# B&R Automation Studio project A2019059_Linka_Power_CP (part 47)

#### Main.st - Init, cyclic, exit code
```iecst
PROGRAM _INIT
	(* Insert code here *)
    SKTcpClientTrace_1.Params.IPportClient := 21001;
END_PROGRAM

PROGRAM _CYCLIC

	//Priradenie indexu paletky//
    a:= P3_LeakageTestB.PAR.IndexPaletky;

    //Parametre komunikácie//
    memcpy(ADR(SKTcpClientTrace_1.Params.IPaddrServ),ADR('192.168.122.250'),SIZEOF('192.168.122.250'));

    SKTcpClientTrace_1.Params.IPportServ := 12000;
    SKTcpClientTrace_1.Params.RecvTimeout := 10000;
    SKTcpClientTrace_1();

    //Parametre komunikácie//
    //Vstupy pre server//
    SKTcpClientTrace_1.Params.Packet.type := TRCB_P3_LeakageTestB_ST8B.INPUTS.TYP_Prikazu;
    SKTcpClientTrace_1.Params.Packet.workplace := TRCB_P3_LeakageTestB_ST8B.INPUTS.CisloStanice;
    TRCB_P3_LeakageTestB_ST8B.INPUTS.CisloPaletky:= 'Pal';
    brsstrcat(ADR(TRCB_P3_LeakageTestB_ST8B.INPUTS.CisloPaletky), ADR(P3_LeakageTestB.PAR.IndexPaletky_STRING));
    SKTcpClientTrace_1.Params.Packet.rfid := TRCB_P3_LeakageTestB_ST8B.INPUTS.CisloPaletky;
    SKTcpClientTrace_1.Params.Packet.master := TRCB_P3_LeakageTestB_ST8B.INPUTS.QRkodPowerCP;
    SKTcpClientTrace_1.Params.Packet.dps1:= TRCB_P3_LeakageTestB_ST8B.INPUTS.QRkodFiltra;
    SKTcpClientTrace_1.Params.Packet.dps2:= '';
    SKTcpClientTrace_1.Params.Packet.dps3:= '';
    SKTcpClientTrace_1.Params.Packet.dps4:= '';
    SKTcpClientTrace_1.Params.Packet.dps5:= '';
    SKTcpClientTrace_1.Params.Packet.operator_id := TRCB_P3_LeakageTestB_ST8B.INPUTS.ID_Operatora;
    SKTcpClientTrace_1.Params.Packet.data_report:= TRCB_P3_LeakageTestB_ST8B.INPUTS.Report;
    SKTcpClientTrace_1.Params.Packet.result := TRCB_P3_LeakageTestB_ST8B.INPUTS.StavPaletky;

    //Výstupy zo servera//
    TRCB_P3_LeakageTestB_ST8B.OUTPUTS.TYP_Prikazu:= SKTcpClientTrace_1.Internal.Splitter.out[1];
    TRCB_P3_LeakageTestB_ST8B.OUTPUTS.CisloStanice:= SKTcpClientTrace_1.Internal.Splitter.out[2];
    TRCB_P3_LeakageTestB_ST8B.OUTPUTS.CisloPaletky:= SKTcpClientTrace_1.Internal.Splitter.out[3];
    IF TRCB_P3_LeakageTestB_ST8B.INPUTS.TYP_Prikazu = '0' THEN
        TRCB_P3_LeakageTestB_ST8B.OUTPUTS.CisloEtikety:= SKTcpClientTrace_1.Internal.Splitter.out[4];
    ELSE
        TRCB_P3_LeakageTestB_ST8B.OUTPUTS.QRkodPowerCP:= SKTcpClientTrace_1.Internal.Splitter.out[4];
    END_IF
    TRCB_P3_LeakageTestB_ST8B.OUTPUTS.QRkodFiltra:= SKTcpClientTrace_1.Internal.Splitter.out[5];
    TRCB_P3_LeakageTestB_ST8B.OUTPUTS.ID_Operatora:= SKTcpClientTrace_1.Internal.Splitter.out[10];
    TRCB_P3_LeakageTestB_ST8B.OUTPUTS.DruhCinnostiNaPaletke:= SKTcpClientTrace_1.Internal.Splitter.out[11];
    TRCB_P3_LeakageTestB_ST8B.OUTPUTS.PovolenieCinnostiNaPaletke:= SKTcpClientTrace_1.Internal.Splitter.out[12];

    //Volanie funkcie SequenceControl//
    SequenceControl(SC:= SC_KOM_Server);

    CASE SC_KOM_Server.Step OF

        0:
            SC_KOM_Server.StepName:= '0 - Nulovanie';
            SKTcpClientTrace_1.Cmd.Send:= FALSE;
            SKTcpClientTrace_1.Cmd.Close:= FALSE;
            TRCB_P3_LeakageTestB_ST8B.CMD.VyziadajStavPaletky_TYP1:= FALSE;
            TRCB_P3_LeakageTestB_ST8B.CMD.PriradQRkodFiltra_TYP3:= FALSE;
            TRCB_P3_LeakageTestB_ST8B.CMD.VyziadajCisloEtikety_TYP0:= FALSE;
            TRCB_P3_LeakageTestB_ST8B.CMD.OdosliStavPaletky_TYP2:= FALSE;
            TRCB_P3_LeakageTestB_ST8B.STATUS.KomunikaciaUkoncena:= FALSE;
            TRCB_P3_LeakageTestB_ST8B.STATUS.KomunikaciaError:= FALSE;
            PocetDopytovNaServer:= 0;

            IF SKTcpClientTrace_1.Internal.Step = 0 THEN
                SKTcpClientTrace_1.Enable:= TRUE;
                SC_KOM_Server.ResetStep:= TRUE;
                SC_KOM_Server.Step:= 1;
            ELSIF SKTcpClientTrace_1.Internal.Step = 15 THEN
                SKTcpClientTrace_1.Enable:= TRUE;
                SC_KOM_Server.ResetStep:= TRUE;
                SC_KOM_Server.Step:= 1;
            ELSE
                SKTcpClientTrace_1.Enable:= FALSE;
            END_IF

        1:
            SC_KOM_Server.StepName:= '1 - Rozhodnutie o cinnosti';
            IF TRCB_P3_LeakageTestB_ST8B.CMD.VyziadajStavPaletky_TYP1 THEN
                SC_KOM_Server.Step:= 10;
            ELSIF TRCB_P3_LeakageTestB_ST8B.CMD.PriradQRkodFiltra_TYP3 THEN
                SC_KOM_Server.Step:= 20;
            ELSIF TRCB_P3_LeakageTestB_ST8B.CMD.VyziadajCisloEtikety_TYP0 THEN
                SC_KOM_Server.Step:= 30;
            ELSIF TRCB_P3_LeakageTestB_ST8B.CMD.OdosliStavPaletky_TYP2 THEN
                SC_KOM_Server.Step:= 40;
            END_IF

        10:
            SC_KOM_Server.StepName:= '10 - Vyziadanie stavu paletky - odoslanie dat na server';
            SC_KOM_Server.IdleTime.PT:= T#3s;
            SC_KOM_Server.AlarmTime.PT:= T#10s;
            SC_KOM_Server.AlarmTime.IN:= TRUE;

            TRCB_P3_LeakageTestB_ST8B.INPUTS.TYP_Prikazu:= '1';
            TRCB_P3_LeakageTestB_ST8B.INPUTS.CisloStanice:= 'ST8B';
            TRCB_P3_LeakageTestB_ST8B.INPUTS.CisloPaletky; //Z programu
            TRCB_P3_LeakageTestB_ST8B.INPUTS.QRkodPowerCP:= Paletka[a].PAR.QRkodPowerCP;
            TRCB_P3_LeakageTestB_ST8B.INPUTS.QRkodFiltra:= '';
            TRCB_P3_LeakageTestB_ST8B.INPUTS.ID_Operatora:= Paletka[a].PAR.ID_Operatora;
            TRCB_P3_LeakageTestB_ST8B.INPUTS.Report:= '';
            TRCB_P3_LeakageTestB_ST8B.INPUTS.StavPaletky:= 'OK';
            SKTcpClientTrace_1.Cmd.Send:= TRUE;

            IF SKTcpClientTrace_1.Cmd.Send AND NOT SKTcpClientTrace_1.Status.staReceived AND NOT SKTcpClientTrace_1.Status.staError THEN
                SC_KOM_Server.ResetStep:= TRUE;
                SC_KOM_Server.Step:= 13;
            ELSIF SC_KOM_Server.AlarmTime.Q AND (SKTcpClientTrace_1.Status.staReceived OR SKTcpClientTrace_1.Status.staError) THEN
                PocetDopytovNaServer:= PocetDopytovNaServer + 1;
                SKTcpClientTrace_1.Cmd.Send:= FALSE;
                SC_KOM_Server.ResetStep:= TRUE;
                SC_KOM_Server.Step:= 14;
            END_IF

        13:
            SC_KOM_Server.StepName:= '13 - Vyziadanie stavu paletky - odpoved servera';
            SC_KOM_Server.IdleTime.PT:= T#3s;
            SC_KOM_Server.AlarmTime.PT:= T#20s;
            SC_KOM_Server.AlarmTime.IN:= TRUE;

            IF SKTcpClientTrace_1.Status.staReceived AND
                (TRCB_P3_LeakageTestB_ST8B.OUTPUTS.TYP_Prikazu = TRCB_P3_LeakageTestB_ST8B.INPUTS.TYP_Prikazu) AND
                (TRCB_P3_LeakageTestB_ST8B.OUTPUTS.QRkodPowerCP = TRCB_P3_LeakageTestB_ST8B.INPUTS.QRkodPowerCP) THEN
                TRCB_P3_LeakageTestB_ST8B.STATUS.KomunikaciaUkoncena:= TRUE;
                SC_KOM_Server.ResetStep:= TRUE;
                SC_KOM_Server.Step:= 15;
            ELSIF SC_KOM_Server.AlarmTime.Q THEN
                PocetDopytovNaServer:= PocetDopytovNaServer + 1;
                SC_KOM_Server.ResetStep:= TRUE;
                SC_KOM_Server.Step:= 14;
            END_IF

        14:
            SC_KOM_Server.StepName:= '14 - Vyziadanie stavu paletky - cakam na opatovny dopyt na server';
            SC_KOM_Server.IdleTime.PT:= T#1s;
            SC_KOM_Server.AlarmTime.PT:= T#10s;
            SC_KOM_Server.IdleTime.IN:= TRUE;

            IF PocetDopytovNaServer < 3 THEN
                IF SC_KOM_Server.IdleTime.Q THEN
                    SC_KOM_Server.ResetStep:= TRUE;
                    SC_KOM_Server.Step:= 10;
                END_IF
            ELSE
                TRCB_P3_LeakageTestB_ST8B.STATUS.KomunikaciaError:= TRUE;
                SC_KOM_Server.ResetStep:= TRUE;
                SC_KOM_Server.Step:= 15;
            END_IF

        15:
            SC_KOM_Server.StepName:= '15 - Vyziadanie stavu paletky - cakam na ukoncenie komunikacie';
            SC_KOM_Server.IdleTime.PT:= T#3s;
            SC_KOM_Server.AlarmTime.PT:= T#10s;

            IF NOT TRCB_P3_LeakageTestB_ST8B.CMD.VyziadajStavPaletky_TYP1 THEN
                SC_KOM_Server.ResetStep:= TRUE;
                SC_KOM_Server.Step:= 0;
            END_IF

        20:
            SC_KOM_Server.StepName:= '20 - Priradenie QR kodu - odoslanie dat na server';
            SC_KOM_Server.IdleTime.PT:= T#3s;
            SC_KOM_Server.AlarmTime.PT:= T#10s;

            TRCB_P3_LeakageTestB_ST8B.INPUTS.TYP_Prikazu:= '3';
            TRCB_P3_LeakageTestB_ST8B.INPUTS.CisloStanice:= 'ST8B';
            TRCB_P3_LeakageTestB_ST8B.INPUTS.CisloPaletky;
            TRCB_P3_LeakageTestB_ST8B.INPUTS.QRkodPowerCP:= Paletka[a].PAR.QRkodPowerCP;
            TRCB_P3_LeakageTestB_ST8B.INPUTS.QRkodFiltra:= '';
            TRCB_P3_LeakageTestB_ST8B.INPUTS.ID_Operatora:= Paletka[a].PAR.ID_Operatora;
            TRCB_P3_LeakageTestB_ST8B.INPUTS.Report:= '';
            TRCB_P3_LeakageTestB_ST8B.INPUTS.StavPaletky:= 'OK';
            SKTcpClientTrace_1.Cmd.Send:= TRUE;

            IF SKTcpClientTrace_1.Cmd.Send AND NOT SKTcpClientTrace_1.Status.staReceived AND NOT SKTcpClientTrace_1.Status.staError THEN
                SC_KOM_Server.ResetStep:= TRUE;
                SC_KOM_Server.Step:= 23;
            END_IF

        23:
            SC_KOM_Server.StepName:= '23 - Priradenie QR kodu - odpoved servera';
            SC_KOM_Server.IdleTime.PT:= T#3s;
            SC_KOM_Server.AlarmTime.PT:= T#20s;
            SC_KOM_Server.AlarmTime.IN:= TRUE;

            IF SKTcpClientTrace_1.Status.staReceived AND
                (TRCB_P3_LeakageTestB_ST8B.OUTPUTS.TYP_Prikazu = TRCB_P3_LeakageTestB_ST8B.INPUTS.TYP_Prikazu) AND
                (TRCB_P3_LeakageTestB_ST8B.OUTPUTS.QRkodPowerCP = TRCB_P3_LeakageTestB_ST8B.INPUTS.QRkodPowerCP) THEN
                TRCB_P3_LeakageTestB_ST8B.STATUS.KomunikaciaUkoncena:= TRUE;
                SC_KOM_Server.ResetStep:= TRUE;
                SC_KOM_Server.Step:= 25;
            ELSIF SC_KOM_Server.AlarmTime.Q THEN
                TRCB_P3_LeakageTestB_ST8B.STATUS.KomunikaciaError:= TRUE;
                SC_KOM_Server.ResetStep:= TRUE;
                SC_KOM_Server.Step:= 25;
            END_IF

        25:
            SC_KOM_Server.StepName:= '25 - Vyziadanie stavu paletky - cakam na ukoncenie komunikacie';
            SC_KOM_Server.IdleTime.PT:= T#3s;
            SC_KOM_Server.AlarmTime.PT:= T#10s;

            IF NOT TRCB_P3_LeakageTestB_ST8B.CMD.PriradQRkodFiltra_TYP3 THEN
                SC_KOM_Server.ResetStep:= TRUE;
                SC_KOM_Server.Step:= 0;
            END_IF

        30:
            SC_KOM_Server.StepName:= '30 - Vyziadanie serioveho cisla - odoslanie dat na server';
            SC_KOM_Server.IdleTime.PT:= T#3s;
            SC_KOM_Server.AlarmTime.PT:= T#10s;

            TRCB_P3_LeakageTestB_ST8B.INPUTS.TYP_Prikazu:= '0';
            TRCB_P3_LeakageTestB_ST8B.INPUTS.CisloStanice:= 'ST8B';
            TRCB_P3_LeakageTestB_ST8B.INPUTS.CisloPaletky;
            TRCB_P3_LeakageTestB_ST8B.INPUTS.QRkodPowerCP:= '';
            TRCB_P3_LeakageTestB_ST8B.INPUTS.QRkodFiltra:= '';
            TRCB_P3_LeakageTestB_ST8B.INPUTS.ID_Operatora:= 'E2';
            TRCB_P3_LeakageTestB_ST8B.INPUTS.Report:= '';
            TRCB_P3_LeakageTestB_ST8B.INPUTS.StavPaletky:= 'OK';
            SKTcpClientTrace_1.Cmd.Send:= TRUE;

            IF SKTcpClientTrace_1.Cmd.Send AND NOT SKTcpClientTrace_1.Status.staReceived AND NOT SKTcpClientTrace_1.Status.staError THEN
                SC_KOM_Server.ResetStep:= TRUE;
                SC_KOM_Server.Step:= 33;
            END_IF

        33:
            SC_KOM_Server.StepName:= '33 - Vyziadanie serioveho cisla - odpoved servera';
            SC_KOM_Server.IdleTime.PT:= T#3s;
            SC_KOM_Server.AlarmTime.PT:= T#20s;
            SC_KOM_Server.AlarmTime.IN:= TRUE;

            IF SKTcpClientTrace_1.Status.staReceived AND
                (TRCB_P3_LeakageTestB_ST8B.OUTPUTS.TYP_Prikazu = TRCB_P3_LeakageTestB_ST8B.INPUTS.TYP_Prikazu) THEN
                TRCB_P3_LeakageTestB_ST8B.STATUS.KomunikaciaUkoncena:= TRUE;
                SC_KOM_Server.ResetStep:= TRUE;
                SC_KOM_Server.Step:= 35;
            ELSIF SC_KOM_Server.AlarmTime.Q THEN
                TRCB_P3_LeakageTestB_ST8B.STATUS.KomunikaciaError:= TRUE;
                SC_KOM_Server.ResetStep:= TRUE;
                SC_KOM_Server.Step:= 35;
            END_IF

        35:
            SC_KOM_Server.StepName:= '35 - Vyziadanie serioveho cisla - cakam na ukoncenie komunikacie';
            SC_KOM_Server.IdleTime.PT:= T#3s;
            SC_KOM_Server.AlarmTime.PT:= T#10s;

            IF NOT TRCB_P3_LeakageTestB_ST8B.CMD.VyziadajCisloEtikety_TYP0 THEN
                SC_KOM_Server.ResetStep:= TRUE;
                SC_KOM_Server.Step:= 0;
            END_IF

        40:
            SC_KOM_Server.StepName:= '40 - Odoslanie stavu paletky - odoslanie dat na server';
            SC_KOM_Server.IdleTime.PT:= T#3s;
            SC_KOM_Server.AlarmTime.PT:= T#20s;
            SC_KOM_Server.AlarmTime.IN:= TRUE;

            //Vytvorenie spravy pre report//
            IF NOT SC_KOM_Server.Switch1 THEN
                brsmemset(ADR(Report),0,SIZEOF(Report));
                brsmemset(ADR(TRCB_P3_LeakageTestB_ST8B.INPUTS.Report), 0, SIZEOF(TRCB_P3_LeakageTestB_ST8B.INPUTS.Report));

				//Čas plnenia//
                Report[0].PoradoveCislo:= '1';
                Report[0].Popis:= 'StanicaB_CasPlnenia';
                Report[0].FormatHodnoty:= '1';
                Report[0].Tolerancia_MIN_Hodnota:= '';
                Report[0].Tolerancia_MAX_Hodnota:= '';
                Report[0].Nominal:= '';
                Report[0].Tolerancia_MIN_Jednotky:= '';
                Report[0].Tolerancia_MAX_Jednotky:= '';
                Report[0].NameranaHodnota:= Reports.LeakageTest.CasPlnenia.StanicaB;
                Report[0].NameranaHodnota_Jednotky:= 's';
                Report[0].VyslednyResult:= Reports.LeakageTest.VyslednyReport.StanicaB;
                SKTcpClientNewCsvEntry(Report[0].PoradoveCislo,Report[0].Popis,Report[0].FormatHodnoty,Report[0].Tolerancia_MIN_Hodnota,Report[0].Tolerancia_MAX_Hodnota,Report[0].Nominal,Report[0].Tolerancia_MIN_Jednotky,Report[0].Tolerancia_MAX_Jednotky,Report[0].NameranaHodnota,Report[0].NameranaHodnota_Jednotky,Report[0].VyslednyResult, ADR(TRCB_P3_LeakageTestB_ST8B.INPUTS.Report));

                //Čas stabilizacie//
                Report[1].PoradoveCislo:= '2';
                Report[1].Popis:= 'StanicaB_CasStabilizacie';
                Report[1].FormatHodnoty:= '1';
                Report[1].Tolerancia_MIN_Hodnota:= '';
                Report[1].Tolerancia_MAX_Hodnota:= '';
                Report[1].Nominal:= '';
                Report[1].Tolerancia_MIN_Jednotky:= '';
                Report[1].Tolerancia_MAX_Jednotky:= '';
                Report[1].NameranaHodnota:= Reports.LeakageTest.CasStabilizacie.StanicaB;
                Report[1].NameranaHodnota_Jednotky:= 's';
                Report[1].VyslednyResult:= Reports.LeakageTest.VyslednyReport.StanicaB;
                SKTcpClientNewCsvEntry(Report[1].PoradoveCislo,Report[1].Popis,Report[1].FormatHodnoty,Report[1].Tolerancia_MIN_Hodnota,Report[1].Tolerancia_MAX_Hodnota,Report[1].Nominal,Report[1].Tolerancia_MIN_Jednotky,Report[1].Tolerancia_MAX_Jednotky,Report[1].NameranaHodnota,Report[1].NameranaHodnota_Jednotky,Report[1].VyslednyResult, ADR(TRCB_P3_LeakageTestB_ST8B.INPUTS.Report));

                //Tlak plnenia//
                Report[2].PoradoveCislo:= '3';
                Report[2].Popis:= 'StanicaB_TlakPlnenia';
                Report[2].FormatHodnoty:= '1';
                Report[2].Tolerancia_MIN_Hodnota:= '';
                Report[2].Tolerancia_MAX_Hodnota:= '';
                Report[2].Nominal:= '';
                Report[2].Tolerancia_MIN_Jednotky:= '';
                Report[2].Tolerancia_MAX_Jednotky:= '';
                Report[2].NameranaHodnota:= Reports.LeakageTest.TlakPlnenia.StanicaB;
                Report[2].NameranaHodnota_Jednotky:= 'mBar';
                Report[2].VyslednyResult:= Reports.LeakageTest.VyslednyReport.StanicaB;
                SKTcpClientNewCsvEntry(Report[2].PoradoveCislo,Report[2].Popis,Report[2].FormatHodnoty,Report[2].Tolerancia_MIN_Hodnota,Report[2].Tolerancia_MAX_Hodnota,Report[2].Nominal,Report[2].Tolerancia_MIN_Jednotky,Report[2].Tolerancia_MAX_Jednotky,Report[2].NameranaHodnota,Report[2].NameranaHodnota_Jednotky,Report[2].VyslednyResult, ADR(TRCB_P3_LeakageTestB_ST8B.INPUTS.Report));

                //Tlak prítlaku//
                Report[3].PoradoveCislo:= '4';
                Report[3].Popis:= 'StanicaB_TlakPritlaku';
                Report[3].FormatHodnoty:= '1';
                Report[3].Tolerancia_MIN_Hodnota:= Reports.LeakageTest.ToleranciaPritlaku_MIN.StanicaB;
                Report[3].Tolerancia_MAX_Hodnota:= Reports.LeakageTest.ToleranciaPritlaku_MAX.StanicaB;
                Report[3].Nominal:= '';
                Report[3].Tolerancia_MIN_Jednotky:= 'Bar';
                Report[3].Tolerancia_MAX_Jednotky:= 'Bar';
                Report[3].NameranaHodnota:= Reports.LeakageTest.TlakPritlaku.StanicaB;
                Report[3].NameranaHodnota_Jednotky:= 'Bar';
                Report[3].VyslednyResult:= Reports.LeakageTest.VyslednyReport.StanicaB;
                SKTcpClientNewCsvEntry(Report[3].PoradoveCislo,Report[3].Popis,Report[3].FormatHodnoty,Report[3].Tolerancia_MIN_Hodnota,Report[3].Tolerancia_MAX_Hodnota,Report[3].Nominal,Report[3].Tolerancia_MIN_Jednotky,Report[3].Tolerancia_MAX_Jednotky,Report[3].NameranaHodnota,Report[3].NameranaHodnota_Jednotky,Report[3].VyslednyResult, ADR(TRCB_P3_LeakageTestB_ST8B.INPUTS.Report));

                //Tlak úniku//
                Report[4].PoradoveCislo:= '5';
                Report[4].Popis:= 'StanicaB_TlakUniku';
                Report[4].FormatHodnoty:= '1';
                Report[4].Tolerancia_MIN_Hodnota:= Reports.LeakageTest.ToleranciaTlakUniku_MIN.StanicaB;
                Report[4].Tolerancia_MAX_Hodnota:= Reports.LeakageTest.ToleranciaTlakUniku_MAX.StanicaB;
                Report[4].Nominal:= '';
                Report[4].Tolerancia_MIN_Jednotky:= 'Pa';
                Report[4].Tolerancia_MAX_Jednotky:= 'Pa';
                Report[4].NameranaHodnota:= Reports.LeakageTest.TlakUniku.StanicaB;
                Report[4].NameranaHodnota_Jednotky:= 'Pa';
                Report[4].VyslednyResult:= Reports.LeakageTest.VyslednyReport.StanicaB;
                SKTcpClientNewCsvEntry(Report[4].PoradoveCislo,Report[4].Popis,Report[4].FormatHodnoty,Report[4].Tolerancia_MIN_Hodnota,Report[4].Tolerancia_MAX_Hodnota,Report[4].Nominal,Report[4].Tolerancia_MIN_Jednotky,Report[4].Tolerancia_MAX_Jednotky,Report[4].NameranaHodnota,Report[4].NameranaHodnota_Jednotky,Report[4].VyslednyResult, ADR(TRCB_P3_LeakageTestB_ST8B.INPUTS.Report));

                //Tolerancia//
                Report[5].PoradoveCislo:= '6';
                Report[5].Popis:= 'StanicaB_Tolerancia';
                Report[5].FormatHodnoty:= '1';
                Report[5].Tolerancia_MIN_Hodnota:= '';
                Report[5].Tolerancia_MAX_Hodnota:= '';
                Report[5].Nominal:= '';
                Report[5].Tolerancia_MIN_Jednotky:= '';
                Report[5].Tolerancia_MAX_Jednotky:= '';
                Report[5].NameranaHodnota:= Reports.LeakageTest.Tolerancia.StanicaB;
                Report[5].NameranaHodnota_Jednotky:= 'Pa';
                Report[5].VyslednyResult:= Reports.LeakageTest.VyslednyReport.StanicaB;
                SKTcpClientNewCsvEntry(Report[5].PoradoveCislo,Report[5].Popis,Report[5].FormatHodnoty,Report[5].Tolerancia_MIN_Hodnota,Report[5].Tolerancia_MAX_Hodnota,Report[5].Nominal,Report[5].Tolerancia_MIN_Jednotky,Report[5].Tolerancia_MAX_Jednotky,Report[5].NameranaHodnota,Report[5].NameranaHodnota_Jednotky,Report[5].VyslednyResult, ADR(TRCB_P3_LeakageTestB_ST8B.INPUTS.Report));

                SC_KOM_Server.Switch1:= TRUE;
            END_IF

            TRCB_P3_LeakageTestB_ST8B.INPUTS.TYP_Prikazu:= '2';
            TRCB_P3_LeakageTestB_ST8B.INPUTS.CisloStanice:= 'ST8B';
            TRCB_P3_LeakageTestB_ST8B.INPUTS.CisloPaletky;
            TRCB_P3_LeakageTestB_ST8B.INPUTS.QRkodPowerCP:= Paletka[a].PAR.QRkodPowerCP;
            TRCB_P3_LeakageTestB_ST8B.INPUTS.QRkodFiltra:= '';
            TRCB_P3_LeakageTestB_ST8B.INPUTS.ID_Operatora:= Paletka[a].PAR.ID_Operatora;
            TRCB_P3_LeakageTestB_ST8B.INPUTS.StavPaletky:= Paletka[a].PAR.StavPowerCP;
            SKTcpClientTrace_1.Cmd.Send:= TRUE;

            IF SKTcpClientTrace_1.Cmd.Send AND NOT SKTcpClientTrace_1.Status.staReceived AND NOT SKTcpClientTrace_1.Status.staError THEN
                SC_KOM_Server.ResetStep:= TRUE;
                SC_KOM_Server.Step:= 43;
            ELSIF SC_KOM_Server.AlarmTime.Q AND (SKTcpClientTrace_1.Status.staReceived OR SKTcpClientTrace_1.Status.staError) THEN
                PocetDopytovNaServer:= PocetDopytovNaServer + 1;
                SC_KOM_Server.ResetStep:= TRUE;
                SC_KOM_Server.Step:= 44;
            END_IF

        43:
            SC_KOM_Server.StepName:= '43 - Odoslanie stavu paletky - odpoved servera';
            SC_KOM_Server.IdleTime.PT:= T#3s;
            SC_KOM_Server.AlarmTime.PT:= T#20s;
            SC_KOM_Server.AlarmTime.IN:= TRUE;

            IF SKTcpClientTrace_1.Status.staReceived AND
                (TRCB_P3_LeakageTestB_ST8B.OUTPUTS.TYP_Prikazu = TRCB_P3_LeakageTestB_ST8B.INPUTS.TYP_Prikazu) AND
                (TRCB_P3_LeakageTestB_ST8B.OUTPUTS.QRkodPowerCP = TRCB_P3_LeakageTestB_ST8B.INPUTS.QRkodPowerCP) THEN
                TRCB_P3_LeakageTestB_ST8B.STATUS.KomunikaciaUkoncena:= TRUE;
                SC_KOM_Server.ResetStep:= TRUE;
                SC_KOM_Server.Step:= 45;
            ELSIF SC_KOM_Server.AlarmTime.Q THEN
                PocetDopytovNaServer:= PocetDopytovNaServer + 1;
                SC_KOM_Server.ResetStep:= TRUE;
                SC_KOM_Server.Step:= 44;
            END_IF

        44:
            SC_KOM_Server.StepName:= '44 - Odoslanie stavu paletky - cakam na opatovny dopyt na server';
            SC_KOM_Server.IdleTime.PT:= T#1s;
            SC_KOM_Server.AlarmTime.PT:= T#10s;
            SC_KOM_Server.IdleTime.IN:= TRUE;
            SKTcpClientTrace_1.Cmd.Send:= FALSE;

            IF PocetDopytovNaServer < 3 THEN
                IF SC_KOM_Server.IdleTime.Q THEN
                    SC_KOM_Server.ResetStep:= TRUE;
                    SC_KOM_Server.Step:= 40;
                END_IF
            ELSE
                TRCB_P3_LeakageTestB_ST8B.STATUS.KomunikaciaError:= TRUE;
                SC_KOM_Server.ResetStep:= TRUE;
                SC_KOM_Server.Step:= 45;
            END_IF

        45:
            SC_KOM_Server.StepName:= '45 - Odoslanie stavu paletky - cakam na ukoncenie komunikacie';
            SC_KOM_Server.IdleTime.PT:= T#3s;
            SC_KOM_Server.AlarmTime.PT:= T#10s;

            IF NOT TRCB_P3_LeakageTestB_ST8B.CMD.OdosliStavPaletky_TYP2 THEN
                SC_KOM_Server.ResetStep:= TRUE;
                SC_KOM_Server.Step:= 0;
            END_IF

    END_CASE

END_PROGRAM

PROGRAM _EXIT
	(* Insert code here *)

END_PROGRAM
```

#### Types.typ - Local data types
```iecst
TYPE
	Report_typ : 	STRUCT
		PoradoveCislo : STRING[2]; (*IDstep - Poradové čislo reportu*)
		Popis : STRING[100]; (*Description - Popis*)
		FormatHodnoty : STRING[2]; (*TypValue - Format zaslané hodnoty  1- Číslo, 2 - Znak*)
		Tolerancia_MIN_Hodnota : STRING[10]; (*MinTol - Minimálna tolerancia meranej veličiny*)
		Tolerancia_MAX_Hodnota : STRING[10]; (*MaxTol - Maximálna tolerancia meranej veličiny*)
		Nominal : STRING[10]; (*Nom - Ak jezvolený formát string tak tu zadáme OK inak je prazdna*)
		Tolerancia_MIN_Jednotky : STRING[10]; (*MinEle - Jednotky minimálnej tolerancie veličiny*)
		Tolerancia_MAX_Jednotky : STRING[10]; (*MaxEle - Jednotky maximálnej tolerancie veličiny*)
		NameranaHodnota : STRING[10]; (*Value - Namerana hodnota veličiny, ak su kamery tak bude hodnota OK alebo NG*)
		NameranaHodnota_Jednotky : STRING[10]; (*ValEle - Jednotky nameranej veličiny*)
		VyslednyResult : STRING[5]; (*Result - Výsledný result  PASS, FAIL, SKIP*)
	END_STRUCT;
END_TYPE
```

#### Variables.var - Local variables
```iecst
VAR
	SC_KOM_Server : SequenceControlTyp;
	SKTcpClientTrace_1 : SKTcpClientTrace;
	a : USINT;
	Report : ARRAY[0..50] OF Report_typ;
	PocetDopytovNaServer : USINT;
END_VAR
```

### Program Logical/TracebilitySystem/P4_Etiketovacka_ST9 (IEC)

#### Main.st - Init, cyclic, exit code
```iecst
PROGRAM _INIT
	(* Insert code here *)
    SKTcpClientTrace_1.Params.IPportClient := 22000;
END_PROGRAM

PROGRAM _CYCLIC

	//Priradenie indexu paletky//
    a:= P4_Etiketovacka.PAR.IndexPaletky;

    //Parametre komunikácie//
    memcpy(ADR(SKTcpClientTrace_1.Params.IPaddrServ),ADR('192.168.122.250'),SIZEOF('192.168.122.250'));

    SKTcpClientTrace_1.Params.IPportServ := 12000;
    SKTcpClientTrace_1.Params.RecvTimeout := 10000;
    SKTcpClientTrace_1();

    //Parametre komunikácie//
    //Vstupy pre server//
    SKTcpClientTrace_1.Params.Packet.type := TRCB_P4_Etiketovacka_ST9.INPUTS.TYP_Prikazu;
    SKTcpClientTrace_1.Params.Packet.workplace := TRCB_P4_Etiketovacka_ST9.INPUTS.CisloStanice;
    TRCB_P4_Etiketovacka_ST9.INPUTS.CisloPaletky:= 'Pal';
    brsstrcat(ADR(TRCB_P4_Etiketovacka_ST9.INPUTS.CisloPaletky), ADR(P4_Etiketovacka.PAR.IndexPaletky_STRING));
    SKTcpClientTrace_1.Params.Packet.rfid := TRCB_P4_Etiketovacka_ST9.INPUTS.CisloPaletky;
    SKTcpClientTrace_1.Params.Packet.master := TRCB_P4_Etiketovacka_ST9.INPUTS.QRkodPowerCP;
    SKTcpClientTrace_1.Params.Packet.dps1:= TRCB_P4_Etiketovacka_ST9.INPUTS.QRkodFiltra;
    SKTcpClientTrace_1.Params.Packet.dps2:= '';
    SKTcpClientTrace_1.Params.Packet.dps3:= '';
    SKTcpClientTrace_1.Params.Packet.dps4:= '';
    SKTcpClientTrace_1.Params.Packet.dps5:= '';
    SKTcpClientTrace_1.Params.Packet.operator_id := TRCB_P4_Etiketovacka_ST9.INPUTS.ID_Operatora;
    SKTcpClientTrace_1.Params.Packet.data_report:= TRCB_P4_Etiketovacka_ST9.INPUTS.Report;
    SKTcpClientTrace_1.Params.Packet.result := TRCB_P4_Etiketovacka_ST9.INPUTS.StavPaletky;

    //Výstupy zo servera//
    TRCB_P4_Etiketovacka_ST9.OUTPUTS.TYP_Prikazu:= SKTcpClientTrace_1.Internal.Splitter.out[1];
    TRCB_P4_Etiketovacka_ST9.OUTPUTS.CisloStanice:= SKTcpClientTrace_1.Internal.Splitter.out[2];
    TRCB_P4_Etiketovacka_ST9.OUTPUTS.CisloPaletky:= SKTcpClientTrace_1.Internal.Splitter.out[3];
    IF TRCB_P4_Etiketovacka_ST9.INPUTS.TYP_Prikazu = '0' THEN
        TRCB_P4_Etiketovacka_ST9.OUTPUTS.CisloEtikety:= SKTcpClientTrace_1.Internal.Splitter.out[4];
    ELSE
        TRCB_P4_Etiketovacka_ST9.OUTPUTS.QRkodPowerCP:= SKTcpClientTrace_1.Internal.Splitter.out[4];
    END_IF
    TRCB_P4_Etiketovacka_ST9.OUTPUTS.QRkodFiltra:= SKTcpClientTrace_1.Internal.Splitter.out[5];
    TRCB_P4_Etiketovacka_ST9.OUTPUTS.ID_Operatora:= SKTcpClientTrace_1.Internal.Splitter.out[10];
    TRCB_P4_Etiketovacka_ST9.OUTPUTS.DruhCinnostiNaPaletke:= SKTcpClientTrace_1.Internal.Splitter.out[11];
    TRCB_P4_Etiketovacka_ST9.OUTPUTS.PovolenieCinnostiNaPaletke:= SKTcpClientTrace_1.Internal.Splitter.out[12];

    //Volanie funkcie SequenceControl//
    SequenceControl(SC:= SC_KOM_Server);

    CASE SC_KOM_Server.Step OF

        0:
            SC_KOM_Server.StepName:= '0 - Nulovanie';
            SKTcpClientTrace_1.Cmd.Send:= FALSE;
            SKTcpClientTrace_1.Cmd.Close:= FALSE;
            TRCB_P4_Etiketovacka_ST9.CMD.VyziadajStavPaletky_TYP1:= FALSE;
            TRCB_P4_Etiketovacka_ST9.CMD.PriradQRkodFiltra_TYP3:= FALSE;
            TRCB_P4_Etiketovacka_ST9.CMD.VyziadajCisloEtikety_TYP0:= FALSE;
            TRCB_P4_Etiketovacka_ST9.CMD.OdosliStavPaletky_TYP2:= FALSE;
            TRCB_P4_Etiketovacka_ST9.STATUS.KomunikaciaUkoncena:= FALSE;
            TRCB_P4_Etiketovacka_ST9.STATUS.KomunikaciaError:= FALSE;
            PocetDopytovNaServer:= 0;

            IF SKTcpClientTrace_1.Internal.Step = 0 THEN
                SKTcpClientTrace_1.Enable:= TRUE;
                SC_KOM_Server.ResetStep:= TRUE;
                SC_KOM_Server.Step:= 1;
            ELSIF SKTcpClientTrace_1.Internal.Step = 15 THEN
                SKTcpClientTrace_1.Enable:= TRUE;
                SC_KOM_Server.ResetStep:= TRUE;
                SC_KOM_Server.Step:= 1;
            ELSE
                SKTcpClientTrace_1.Enable:= FALSE;
            END_IF

        1:
            SC_KOM_Server.StepName:= '1 - Rozhodnutie o cinnosti';
            IF TRCB_P4_Etiketovacka_ST9.CMD.VyziadajStavPaletky_TYP1 THEN
                SC_KOM_Server.Step:= 10;
            ELSIF TRCB_P4_Etiketovacka_ST9.CMD.PriradQRkodFiltra_TYP3 THEN
                SC_KOM_Server.Step:= 20;
            ELSIF TRCB_P4_Etiketovacka_ST9.CMD.VyziadajCisloEtikety_TYP0 THEN
                SC_KOM_Server.Step:= 30;
            ELSIF TRCB_P4_Etiketovacka_ST9.CMD.OdosliStavPaletky_TYP2 THEN
                SC_KOM_Server.Step:= 40;
            END_IF

        10:
            SC_KOM_Server.StepName:= '10 - Vyziadanie stavu paletky - odoslanie dat na server';
            SC_KOM_Server.IdleTime.PT:= T#3s;
            SC_KOM_Server.AlarmTime.PT:= T#10s;
            SC_KOM_Server.AlarmTime.IN:= TRUE;

            TRCB_P4_Etiketovacka_ST9.INPUTS.TYP_Prikazu:= '1';
            TRCB_P4_Etiketovacka_ST9.INPUTS.CisloStanice:= 'ST9';
            TRCB_P4_Etiketovacka_ST9.INPUTS.CisloPaletky; //Z programu
            TRCB_P4_Etiketovacka_ST9.INPUTS.QRkodPowerCP:= Paletka[a].PAR.QRkodPowerCP;
            TRCB_P4_Etiketovacka_ST9.INPUTS.QRkodFiltra:= '';
            TRCB_P4_Etiketovacka_ST9.INPUTS.ID_Operatora:= Paletka[a].PAR.ID_Operatora;
            TRCB_P4_Etiketovacka_ST9.INPUTS.Report:= '';
            TRCB_P4_Etiketovacka_ST9.INPUTS.StavPaletky:= 'OK';
            SKTcpClientTrace_1.Cmd.Send:= TRUE;

            IF SKTcpClientTrace_1.Cmd.Send AND NOT SKTcpClientTrace_1.Status.staReceived AND NOT SKTcpClientTrace_1.Status.staError THEN
                SC_KOM_Server.ResetStep:= TRUE;
                SC_KOM_Server.Step:= 13;
            ELSIF SC_KOM_Server.AlarmTime.Q AND (SKTcpClientTrace_1.Status.staReceived OR SKTcpClientTrace_1.Status.staError) THEN
                PocetDopytovNaServer:= PocetDopytovNaServer + 1;
                SKTcpClientTrace_1.Cmd.Send:= FALSE;
                SC_KOM_Server.ResetStep:= TRUE;
                SC_KOM_Server.Step:= 14;
            END_IF

        13:
            SC_KOM_Server.StepName:= '13 - Vyziadanie stavu paletky - odpoved servera';
            SC_KOM_Server.IdleTime.PT:= T#3s;
            SC_KOM_Server.AlarmTime.PT:= T#20s;
            SC_KOM_Server.AlarmTime.IN:= TRUE;

            IF SKTcpClientTrace_1.Status.staReceived AND
                (TRCB_P4_Etiketovacka_ST9.OUTPUTS.TYP_Prikazu = TRCB_P4_Etiketovacka_ST9.INPUTS.TYP_Prikazu) AND
                (TRCB_P4_Etiketovacka_ST9.OUTPUTS.QRkodPowerCP = TRCB_P4_Etiketovacka_ST9.INPUTS.QRkodPowerCP) THEN
                TRCB_P4_Etiketovacka_ST9.STATUS.KomunikaciaUkoncena:= TRUE;
                SC_KOM_Server.ResetStep:= TRUE;
                SC_KOM_Server.Step:= 15;
            ELSIF SC_KOM_Server.AlarmTime.Q THEN
                PocetDopytovNaServer:= PocetDopytovNaServer + 1;
                SC_KOM_Server.ResetStep:= TRUE;
                SC_KOM_Server.Step:= 14;
            END_IF

        14:
            SC_KOM_Server.StepName:= '14 - Vyziadanie stavu paletky - cakam na opatovny dopyt na server';
            SC_KOM_Server.IdleTime.PT:= T#1s;
            SC_KOM_Server.AlarmTime.PT:= T#10s;
            SC_KOM_Server.IdleTime.IN:= TRUE;

            IF PocetDopytovNaServer < 3 THEN
                IF SC_KOM_Server.IdleTime.Q THEN
                    SC_KOM_Server.ResetStep:= TRUE;
                    SC_KOM_Server.Step:= 10;
                END_IF
            ELSE
                TRCB_P4_Etiketovacka_ST9.STATUS.KomunikaciaError:= TRUE;
                SC_KOM_Server.ResetStep:= TRUE;
                SC_KOM_Server.Step:= 15;
            END_IF

        15:
            SC_KOM_Server.StepName:= '15 - Vyziadanie stavu paletky - cakam na ukoncenie komunikacie';
            SC_KOM_Server.IdleTime.PT:= T#3s;
            SC_KOM_Server.AlarmTime.PT:= T#10s;

            IF NOT TRCB_P4_Etiketovacka_ST9.CMD.VyziadajStavPaletky_TYP1 THEN
                SC_KOM_Server.ResetStep:= TRUE;
                SC_KOM_Server.Step:= 0;
            END_IF

        20:
            SC_KOM_Server.StepName:= '20 - Priradenie QR kodu - odoslanie dat na server';
            SC_KOM_Server.IdleTime.PT:= T#3s;
            SC_KOM_Server.AlarmTime.PT:= T#10s;

            TRCB_P4_Etiketovacka_ST9.INPUTS.TYP_Prikazu:= '3';
            TRCB_P4_Etiketovacka_ST9.INPUTS.CisloStanice:= 'ST9';
            TRCB_P4_Etiketovacka_ST9.INPUTS.CisloPaletky;
            TRCB_P4_Etiketovacka_ST9.INPUTS.QRkodPowerCP:= Paletka[a].PAR.QRkodPowerCP;
            TRCB_P4_Etiketovacka_ST9.INPUTS.QRkodFiltra:= '';
            TRCB_P4_Etiketovacka_ST9.INPUTS.ID_Operatora:= Paletka[a].PAR.ID_Operatora;
            TRCB_P4_Etiketovacka_ST9.INPUTS.Report:= '';
            TRCB_P4_Etiketovacka_ST9.INPUTS.StavPaletky:= 'OK';
            SKTcpClientTrace_1.Cmd.Send:= TRUE;

            IF SKTcpClientTrace_1.Cmd.Send AND NOT SKTcpClientTrace_1.Status.staReceived AND NOT SKTcpClientTrace_1.Status.staError THEN
                SC_KOM_Server.ResetStep:= TRUE;
                SC_KOM_Server.Step:= 23;
            END_IF

        23:
            SC_KOM_Server.StepName:= '23 - Priradenie QR kodu - odpoved servera';
            SC_KOM_Server.IdleTime.PT:= T#3s;
            SC_KOM_Server.AlarmTime.PT:= T#20s;
            SC_KOM_Server.AlarmTime.IN:= TRUE;

            IF SKTcpClientTrace_1.Status.staReceived AND
                (TRCB_P4_Etiketovacka_ST9.OUTPUTS.TYP_Prikazu = TRCB_P4_Etiketovacka_ST9.INPUTS.TYP_Prikazu) AND
                (TRCB_P4_Etiketovacka_ST9.OUTPUTS.QRkodPowerCP = TRCB_P4_Etiketovacka_ST9.INPUTS.QRkodPowerCP) THEN
                TRCB_P4_Etiketovacka_ST9.STATUS.KomunikaciaUkoncena:= TRUE;
                SC_KOM_Server.ResetStep:= TRUE;
                SC_KOM_Server.Step:= 25;
            ELSIF SC_KOM_Server.AlarmTime.Q THEN
                TRCB_P4_Etiketovacka_ST9.STATUS.KomunikaciaError:= TRUE;
                SC_KOM_Server.ResetStep:= TRUE;
                SC_KOM_Server.Step:= 25;
            END_IF

        25:
            SC_KOM_Server.StepName:= '25 - Priradenie QR kodu - cakam na ukoncenie komunikacie';
            SC_KOM_Server.IdleTime.PT:= T#3s;
            SC_KOM_Server.AlarmTime.PT:= T#10s;

            IF NOT TRCB_P4_Etiketovacka_ST9.CMD.PriradQRkodFiltra_TYP3 THEN
                SC_KOM_Server.ResetStep:= TRUE;
                SC_KOM_Server.Step:= 0;
            END_IF

        30:
            SC_KOM_Server.StepName:= '30 - Vyziadanie serioveho cisla - odoslanie dat na server';
            SC_KOM_Server.IdleTime.PT:= T#3s;
            SC_KOM_Server.AlarmTime.PT:= T#20s;
            SC_KOM_Server.AlarmTime.IN:= TRUE;

            TRCB_P4_Etiketovacka_ST9.INPUTS.TYP_Prikazu:= '0';
            TRCB_P4_Etiketovacka_ST9.INPUTS.CisloStanice:= 'ST9';
            TRCB_P4_Etiketovacka_ST9.INPUTS.CisloPaletky;
            TRCB_P4_Etiketovacka_ST9.INPUTS.QRkodPowerCP:= '';
            TRCB_P4_Etiketovacka_ST9.INPUTS.QRkodFiltra:= '';
            TRCB_P4_Etiketovacka_ST9.INPUTS.ID_Operatora:= Paletka[a].PAR.ID_Operatora;
            TRCB_P4_Etiketovacka_ST9.INPUTS.Report:= '';
            TRCB_P4_Etiketovacka_ST9.INPUTS.StavPaletky:= 'OK';
            SKTcpClientTrace_1.Cmd.Send:= TRUE;

            IF SKTcpClientTrace_1.Cmd.Send AND NOT SKTcpClientTrace_1.Status.staReceived AND NOT SKTcpClientTrace_1.Status.staError THEN
                SC_KOM_Server.ResetStep:= TRUE;
                SC_KOM_Server.Step:= 33;
            ELSIF SC_KOM_Server.AlarmTime.Q AND (SKTcpClientTrace_1.Status.staReceived OR SKTcpClientTrace_1.Status.staError) THEN
                PocetDopytovNaServer:= PocetDopytovNaServer + 1;
                SC_KOM_Server.ResetStep:= TRUE;
                SC_KOM_Server.Step:= 34;
            END_IF

        33:
            SC_KOM_Server.StepName:= '33 - Vyziadanie serioveho cisla - odpoved servera';
            SC_KOM_Server.IdleTime.PT:= T#3s;
            SC_KOM_Server.AlarmTime.PT:= T#20s;
            SC_KOM_Server.AlarmTime.IN:= TRUE;

            IF SKTcpClientTrace_1.Status.staReceived AND
                (TRCB_P4_Etiketovacka_ST9.OUTPUTS.TYP_Prikazu = TRCB_P4_Etiketovacka_ST9.INPUTS.TYP_Prikazu) THEN
                TRCB_P4_Etiketovacka_ST9.STATUS.KomunikaciaUkoncena:= TRUE;
                SC_KOM_Server.ResetStep:= TRUE;
                SC_KOM_Server.Step:= 35;
            ELSIF SC_KOM_Server.AlarmTime.Q THEN
                PocetDopytovNaServer:= PocetDopytovNaServer + 1;
                SC_KOM_Server.ResetStep:= TRUE;
                SC_KOM_Server.Step:= 34;
            END_IF

        34:
            SC_KOM_Server.StepName:= '34 - Vyziadanie serioveho cisla - cakam na opatovny dopyt na server';
            SC_KOM_Server.IdleTime.PT:= T#1s;
            SC_KOM_Server.AlarmTime.PT:= T#10s;
            SC_KOM_Server.IdleTime.IN:= TRUE;
            SKTcpClientTrace_1.Cmd.Send:= FALSE;

            IF PocetDopytovNaServer < 3 THEN
                IF SC_KOM_Server.IdleTime.Q THEN
                    SC_KOM_Server.ResetStep:= TRUE;
                    SC_KOM_Server.Step:= 30;
                END_IF
            ELSE
                TRCB_P4_Etiketovacka_ST9.STATUS.KomunikaciaError:= TRUE;
                SC_KOM_Server.ResetStep:= TRUE;
                SC_KOM_Server.Step:= 35;
            END_IF

        35:
            SC_KOM_Server.StepName:= '35 - Vyziadanie serioveho cisla - cakam na ukoncenie komunikacie';
            SC_KOM_Server.IdleTime.PT:= T#3s;
            SC_KOM_Server.AlarmTime.PT:= T#10s;

            IF NOT TRCB_P4_Etiketovacka_ST9.CMD.VyziadajCisloEtikety_TYP0 THEN
                SC_KOM_Server.ResetStep:= TRUE;
                SC_KOM_Server.Step:= 0;
            END_IF

        40:
            SC_KOM_Server.StepName:= '40 - Odoslanie stavu paletky - odoslanie dat na server';
            SC_KOM_Server.IdleTime.PT:= T#3s;
            SC_KOM_Server.AlarmTime.PT:= T#20s;
            SC_KOM_Server.AlarmTime.IN:= TRUE;

            IF NOT SC_KOM_Server.Switch1 THEN
                brsmemset(ADR(Report),0,SIZEOF(Report));
               	brsmemset(ADR(TRCB_P4_Etiketovacka_ST9.INPUTS.Report), 0, SIZEOF(TRCB_P4_Etiketovacka_ST9.INPUTS.Report));

				//Kamera 15//
                Report[0].PoradoveCislo:= '1';
                Report[0].Popis:= 'KAM_15_KontrolaEtikety';
                Report[0].FormatHodnoty:= '2';
                Report[0].Tolerancia_MIN_Hodnota:= '';
                Report[0].Tolerancia_MAX_Hodnota:= '';
                Report[0].Nominal:= 'OK';
                Report[0].Tolerancia_MIN_Jednotky:= '';
                Report[0].Tolerancia_MAX_Jednotky:= '';
                IF Reports.Kamery.P4_CAM15_KontrolaPaletky = 'PASS' THEN
                    Report[0].NameranaHodnota:= 'OK';
                ELSE
                    Report[0].NameranaHodnota:= 'NG';
                END_IF
                Report[0].NameranaHodnota_Jednotky:= '';
                Report[0].VyslednyResult:= Reports.Kamery.P4_CAM15_KontrolaPaletky;
                SKTcpClientNewCsvEntry(Report[0].PoradoveCislo,Report[0].Popis,Report[0].FormatHodnoty,Report[0].Tolerancia_MIN_Hodnota,Report[0].Tolerancia_MAX_Hodnota,Report[0].Nominal,Report[0].Tolerancia_MIN_Jednotky,Report[0].Tolerancia_MAX_Jednotky,Report[0].NameranaHodnota,Report[0].NameranaHodnota_Jednotky,Report[0].VyslednyResult, ADR(TRCB_P4_Etiketovacka_ST9.INPUTS.Report));
                SC_KOM_Server.Switch1:= TRUE;
            END_IF

            TRCB_P4_Etiketovacka_ST9.INPUTS.TYP_Prikazu:= '2';
            TRCB_P4_Etiketovacka_ST9.INPUTS.CisloStanice:= 'ST9';
            TRCB_P4_Etiketovacka_ST9.INPUTS.CisloPaletky;
            TRCB_P4_Etiketovacka_ST9.INPUTS.QRkodPowerCP:= Paletka[a].PAR.QRkodPowerCP;
            TRCB_P4_Etiketovacka_ST9.INPUTS.QRkodFiltra:= '';
            TRCB_P4_Etiketovacka_ST9.INPUTS.ID_Operatora:= Paletka[a].PAR.ID_Operatora;
            TRCB_P4_Etiketovacka_ST9.INPUTS.StavPaletky:= Paletka[a].PAR.StavPowerCP;
            SKTcpClientTrace_1.Cmd.Send:= TRUE;

            IF SKTcpClientTrace_1.Cmd.Send AND NOT SKTcpClientTrace_1.Status.staReceived AND NOT SKTcpClientTrace_1.Status.staError THEN
                SC_KOM_Server.ResetStep:= TRUE;
                SC_KOM_Server.Step:= 43;
            ELSIF SC_KOM_Server.AlarmTime.Q AND (SKTcpClientTrace_1.Status.staReceived OR SKTcpClientTrace_1.Status.staError) THEN
                PocetDopytovNaServer:= PocetDopytovNaServer + 1;
                SC_KOM_Server.ResetStep:= TRUE;
                SC_KOM_Server.Step:= 44;
            END_IF

        43:
            SC_KOM_Server.StepName:= '43 - Odoslanie stavu paletky - odpoved servera';
            SC_KOM_Server.IdleTime.PT:= T#3s;
            SC_KOM_Server.AlarmTime.PT:= T#20s;
            SC_KOM_Server.AlarmTime.IN:= TRUE;

            IF SKTcpClientTrace_1.Status.staReceived AND
                (TRCB_P4_Etiketovacka_ST9.OUTPUTS.TYP_Prikazu = TRCB_P4_Etiketovacka_ST9.INPUTS.TYP_Prikazu) AND
                (TRCB_P4_Etiketovacka_ST9.OUTPUTS.QRkodPowerCP = TRCB_P4_Etiketovacka_ST9.INPUTS.QRkodPowerCP) THEN
                TRCB_P4_Etiketovacka_ST9.STATUS.KomunikaciaUkoncena:= TRUE;
                SC_KOM_Server.ResetStep:= TRUE;
                SC_KOM_Server.Step:= 45;
            ELSIF SC_KOM_Server.AlarmTime.Q THEN
                PocetDopytovNaServer:= PocetDopytovNaServer + 1;
                SC_KOM_Server.ResetStep:= TRUE;
                SC_KOM_Server.Step:= 44;
            END_IF

        44:
            SC_KOM_Server.StepName:= '44 - Odoslanie stavu paletky - cakam na opatovny dopyt na server';
            SC_KOM_Server.IdleTime.PT:= T#1s;
            SC_KOM_Server.AlarmTime.PT:= T#10s;
            SC_KOM_Server.IdleTime.IN:= TRUE;
            SKTcpClientTrace_1.Cmd.Send:= FALSE;

            IF PocetDopytovNaServer < 3 THEN
                IF SC_KOM_Server.IdleTime.Q THEN
                    SC_KOM_Server.ResetStep:= TRUE;
                    SC_KOM_Server.Step:= 40;
                END_IF
            ELSE
                TRCB_P4_Etiketovacka_ST9.STATUS.KomunikaciaError:= TRUE;
                SC_KOM_Server.ResetStep:= TRUE;
                SC_KOM_Server.Step:= 45;
            END_IF

        45:
            SC_KOM_Server.StepName:= '45 - Odoslanie stavu paletky - cakam na ukoncenie komunikacie';
            SC_KOM_Server.IdleTime.PT:= T#3s;
            SC_KOM_Server.AlarmTime.PT:= T#10s;

            IF NOT TRCB_P4_Etiketovacka_ST9.CMD.OdosliStavPaletky_TYP2 THEN
                SC_KOM_Server.ResetStep:= TRUE;
                SC_KOM_Server.Step:= 0;
            END_IF

    END_CASE

END_PROGRAM

PROGRAM _EXIT
	(* Insert code here *)

END_PROGRAM
```

#### Types.typ - Local data types
```iecst
TYPE
	Report_typ : 	STRUCT
		PoradoveCislo : STRING[2]; (*IDstep - Poradové čislo reportu*)
		Popis : STRING[100]; (*Description - Popis*)
		FormatHodnoty : STRING[2]; (*TypValue - Format zaslané hodnoty  1- Číslo, 2 - Znak*)
		Tolerancia_MIN_Hodnota : STRING[10]; (*MinTol - Minimálna tolerancia meranej veličiny*)
		Tolerancia_MAX_Hodnota : STRING[10]; (*MaxTol - Maximálna tolerancia meranej veličiny*)
		Nominal : STRING[10]; (*Nom - Ak jezvolený formát string tak tu zadáme OK inak je prazdna*)
		Tolerancia_MIN_Jednotky : STRING[10]; (*MinEle - Jednotky minimálnej tolerancie veličiny*)
		Tolerancia_MAX_Jednotky : STRING[10]; (*MaxEle - Jednotky maximálnej tolerancie veličiny*)
		NameranaHodnota : STRING[10]; (*Value - Namerana hodnota veličiny, ak su kamery tak bude hodnota OK alebo NG*)
		NameranaHodnota_Jednotky : STRING[10]; (*ValEle - Jednotky nameranej veličiny*)
		VyslednyResult : STRING[5]; (*Result - Výsledný result  PASS, FAIL, SKIP*)
	END_STRUCT;
END_TYPE
```

#### Variables.var - Local variables
```iecst
VAR
	SC_KOM_Server : SequenceControlTyp;
	SKTcpClientTrace_1 : SKTcpClientTrace;
	a : USINT;
	Report : ARRAY[0..50] OF Report_typ;
	PocetDopytovNaServer : USINT;
END_VAR
```

### Program Logical/TracebilitySystem/P4_Vytah_ST10 (IEC)

#### Main.st - Init, cyclic, exit code
```iecst
PROGRAM _INIT
	(* Insert code here *)
    SKTcpClientTrace_1.Params.IPportClient := 23000;
END_PROGRAM

PROGRAM _CYCLIC

	//Priradenie indexu paletky//
    a:= P4_Vytah.PAR.IndexPaletky;

    //Parametre komunikácie//
    memcpy(ADR(SKTcpClientTrace_1.Params.IPaddrServ),ADR('192.168.122.250'),SIZEOF('192.168.122.250'));

    SKTcpClientTrace_1.Params.IPportServ := 12000;
    SKTcpClientTrace_1.Params.RecvTimeout := 10000;
    SKTcpClientTrace_1();

    //Parametre komunikácie//
    //Vstupy pre server//
    SKTcpClientTrace_1.Params.Packet.type := TRCB_P4_Vytah_ST10.INPUTS.TYP_Prikazu;
    SKTcpClientTrace_1.Params.Packet.workplace := TRCB_P4_Vytah_ST10.INPUTS.CisloStanice;
    TRCB_P4_Vytah_ST10.INPUTS.CisloPaletky:= 'Pal';
    brsstrcat(ADR(TRCB_P4_Vytah_ST10.INPUTS.CisloPaletky), ADR(P4_Vytah.PAR.IndexPaletky_STRING));
    SKTcpClientTrace_1.Params.Packet.rfid := TRCB_P4_Vytah_ST10.INPUTS.CisloPaletky;
    SKTcpClientTrace_1.Params.Packet.master := TRCB_P4_Vytah_ST10.INPUTS.QRkodPowerCP;
    SKTcpClientTrace_1.Params.Packet.dps1:= TRCB_P4_Vytah_ST10.INPUTS.QRkodFiltra;
    SKTcpClientTrace_1.Params.Packet.dps2:= '';
    SKTcpClientTrace_1.Params.Packet.dps3:= '';
    SKTcpClientTrace_1.Params.Packet.dps4:= '';
    SKTcpClientTrace_1.Params.Packet.dps5:= '';
    SKTcpClientTrace_1.Params.Packet.operator_id := TRCB_P4_Vytah_ST10.INPUTS.ID_Operatora;
    SKTcpClientTrace_1.Params.Packet.data_report:= TRCB_P4_Vytah_ST10.INPUTS.Report;
    SKTcpClientTrace_1.Params.Packet.result := TRCB_P4_Vytah_ST10.INPUTS.StavPaletky;

    //Výstupy zo servera//
    TRCB_P4_Vytah_ST10.OUTPUTS.TYP_Prikazu:= SKTcpClientTrace_1.Internal.Splitter.out[1];
    TRCB_P4_Vytah_ST10.OUTPUTS.CisloStanice:= SKTcpClientTrace_1.Internal.Splitter.out[2];
    TRCB_P4_Vytah_ST10.OUTPUTS.CisloPaletky:= SKTcpClientTrace_1.Internal.Splitter.out[3];
    IF TRCB_P4_Vytah_ST10.INPUTS.TYP_Prikazu = '0' THEN
        TRCB_P4_Vytah_ST10.OUTPUTS.CisloEtikety:= SKTcpClientTrace_1.Internal.Splitter.out[4];
    ELSE
        TRCB_P4_Vytah_ST10.OUTPUTS.QRkodPowerCP:= SKTcpClientTrace_1.Internal.Splitter.out[4];
    END_IF
    TRCB_P4_Vytah_ST10.OUTPUTS.QRkodFiltra:= SKTcpClientTrace_1.Internal.Splitter.out[5];
    TRCB_P4_Vytah_ST10.OUTPUTS.ID_Operatora:= SKTcpClientTrace_1.Internal.Splitter.out[10];
    TRCB_P4_Vytah_ST10.OUTPUTS.DruhCinnostiNaPaletke:= SKTcpClientTrace_1.Internal.Splitter.out[11];
    TRCB_P4_Vytah_ST10.OUTPUTS.PovolenieCinnostiNaPaletke:= SKTcpClientTrace_1.Internal.Splitter.out[12];

    //Volanie funkcie SequenceControl//
    SequenceControl(SC:= SC_KOM_Server);

    CASE SC_KOM_Server.Step OF

        0:
            SC_KOM_Server.StepName:= '0 - Nulovanie';
            SKTcpClientTrace_1.Cmd.Send:= FALSE;
            SKTcpClientTrace_1.Cmd.Close:= FALSE;
            TRCB_P4_Vytah_ST10.CMD.VyziadajStavPaletky_TYP1:= FALSE;
            TRCB_P4_Vytah_ST10.CMD.PriradQRkodFiltra_TYP3:= FALSE;
            TRCB_P4_Vytah_ST10.CMD.VyziadajCisloEtikety_TYP0:= FALSE;
            TRCB_P4_Vytah_ST10.CMD.OdosliStavPaletky_TYP2:= FALSE;
            TRCB_P4_Vytah_ST10.STATUS.KomunikaciaUkoncena:= FALSE;
            TRCB_P4_Vytah_ST10.STATUS.KomunikaciaError:= FALSE;
            PocetDopytovNaServer:= 0;

            IF SKTcpClientTrace_1.Internal.Step = 0 THEN
                SKTcpClientTrace_1.Enable:= TRUE;
                SC_KOM_Server.ResetStep:= TRUE;
                SC_KOM_Server.Step:= 1;
            ELSIF SKTcpClientTrace_1.Internal.Step = 15 THEN
                SKTcpClientTrace_1.Enable:= TRUE;
                SC_KOM_Server.ResetStep:= TRUE;
                SC_KOM_Server.Step:= 1;
            ELSE
                SKTcpClientTrace_1.Enable:= FALSE;
            END_IF

        1:
            SC_KOM_Server.StepName:= '1 - Rozhodnutie o cinnosti';
            IF TRCB_P4_Vytah_ST10.CMD.VyziadajStavPaletky_TYP1 THEN
                SC_KOM_Server.Step:= 10;
            ELSIF TRCB_P4_Vytah_ST10.CMD.PriradQRkodFiltra_TYP3 THEN
                SC_KOM_Server.Step:= 20;
            ELSIF TRCB_P4_Vytah_ST10.CMD.VyziadajCisloEtikety_TYP0 THEN
                SC_KOM_Server.Step:= 30;
            ELSIF TRCB_P4_Vytah_ST10.CMD.OdosliStavPaletky_TYP2 THEN
                SC_KOM_Server.Step:= 40;
            END_IF

        10:
            SC_KOM_Server.StepName:= '10 - Vyziadanie stavu paletky - odoslanie dat na server';
            SC_KOM_Server.IdleTime.PT:= T#3s;
            SC_KOM_Server.AlarmTime.PT:= T#10s;
            SC_KOM_Server.AlarmTime.IN:= TRUE;

            TRCB_P4_Vytah_ST10.INPUTS.TYP_Prikazu:= '1';
            TRCB_P4_Vytah_ST10.INPUTS.CisloStanice:= 'ST10';
            TRCB_P4_Vytah_ST10.INPUTS.CisloPaletky; //Z programu
            TRCB_P4_Vytah_ST10.INPUTS.QRkodPowerCP:= Paletka[a].PAR.QRkodPowerCP;
            TRCB_P4_Vytah_ST10.INPUTS.QRkodFiltra:= '';
            TRCB_P4_Vytah_ST10.INPUTS.ID_Operatora:= Paletka[a].PAR.ID_Operatora;
            TRCB_P4_Vytah_ST10.INPUTS.Report:= '';
            TRCB_P4_Vytah_ST10.INPUTS.StavPaletky:= 'OK';
            SKTcpClientTrace_1.Cmd.Send:= TRUE;

            IF SKTcpClientTrace_1.Cmd.Send AND NOT SKTcpClientTrace_1.Status.staReceived AND NOT SKTcpClientTrace_1.Status.staError THEN
                SC_KOM_Server.ResetStep:= TRUE;
                SC_KOM_Server.Step:= 13;
            ELSIF SC_KOM_Server.AlarmTime.Q AND (SKTcpClientTrace_1.Status.staReceived OR SKTcpClientTrace_1.Status.staError) THEN
                PocetDopytovNaServer:= PocetDopytovNaServer + 1;
                SKTcpClientTrace_1.Cmd.Send:= FALSE;
                SC_KOM_Server.ResetStep:= TRUE;
                SC_KOM_Server.Step:= 14;
            END_IF

        13:
            SC_KOM_Server.StepName:= '13 - Vyziadanie stavu paletky - odpoved servera';
            SC_KOM_Server.IdleTime.PT:= T#3s;
            SC_KOM_Server.AlarmTime.PT:= T#20s;
            SC_KOM_Server.AlarmTime.IN:= TRUE;

            IF SKTcpClientTrace_1.Status.staReceived AND
                (TRCB_P4_Vytah_ST10.OUTPUTS.TYP_Prikazu = TRCB_P4_Vytah_ST10.INPUTS.TYP_Prikazu) AND
                (TRCB_P4_Vytah_ST10.OUTPUTS.QRkodPowerCP = TRCB_P4_Vytah_ST10.INPUTS.QRkodPowerCP) THEN
                TRCB_P4_Vytah_ST10.STATUS.KomunikaciaUkoncena:= TRUE;
                SC_KOM_Server.ResetStep:= TRUE;
                SC_KOM_Server.Step:= 15;
            ELSIF SC_KOM_Server.AlarmTime.Q THEN
                PocetDopytovNaServer:= PocetDopytovNaServer + 1;
                SC_KOM_Server.ResetStep:= TRUE;
                SC_KOM_Server.Step:= 14;
            END_IF

        14:
            SC_KOM_Server.StepName:= '14 - Vyziadanie stavu paletky - cakam na opatovny dopyt na server';
            SC_KOM_Server.IdleTime.PT:= T#1s;
            SC_KOM_Server.AlarmTime.PT:= T#10s;
            SC_KOM_Server.IdleTime.IN:= TRUE;

            IF PocetDopytovNaServer < 3 THEN
                IF SC_KOM_Server.IdleTime.Q THEN
                    SC_KOM_Server.ResetStep:= TRUE;
                    SC_KOM_Server.Step:= 10;
                END_IF
            ELSE
                TRCB_P4_Vytah_ST10.STATUS.KomunikaciaError:= TRUE;
                SC_KOM_Server.ResetStep:= TRUE;
                SC_KOM_Server.Step:= 15;
            END_IF

        15:
            SC_KOM_Server.StepName:= '15 - Vyziadanie stavu paletky - cakam na ukoncenie komunikacie';
            SC_KOM_Server.IdleTime.PT:= T#3s;
            SC_KOM_Server.AlarmTime.PT:= T#10s;

            IF NOT TRCB_P4_Vytah_ST10.CMD.VyziadajStavPaletky_TYP1 THEN
                SC_KOM_Server.ResetStep:= TRUE;
                SC_KOM_Server.Step:= 0;
            END_IF

        20:
            SC_KOM_Server.StepName:= '20 - Priradenie QR kodu - odoslanie dat na server';
            SC_KOM_Server.IdleTime.PT:= T#3s;
            SC_KOM_Server.AlarmTime.PT:= T#10s;

            TRCB_P4_Vytah_ST10.INPUTS.TYP_Prikazu:= '3';
            TRCB_P4_Vytah_ST10.INPUTS.CisloStanice:= 'ST10';
            TRCB_P4_Vytah_ST10.INPUTS.CisloPaletky;
            TRCB_P4_Vytah_ST10.INPUTS.QRkodPowerCP:= Paletka[a].PAR.QRkodPowerCP;
            TRCB_P4_Vytah_ST10.INPUTS.QRkodFiltra:= Paletka[a].PAR.QRkodFiltra_4F5F;
            TRCB_P4_Vytah_ST10.INPUTS.ID_Operatora:= Paletka[a].PAR.ID_Operatora;
            TRCB_P4_Vytah_ST10.INPUTS.Report:= '';
            TRCB_P4_Vytah_ST10.INPUTS.StavPaletky:= 'OK';
            SKTcpClientTrace_1.Cmd.Send:= TRUE;

            IF SKTcpClientTrace_1.Cmd.Send AND NOT SKTcpClientTrace_1.Status.staReceived AND NOT SKTcpClientTrace_1.Status.staError THEN
                SC_KOM_Server.ResetStep:= TRUE;
                SC_KOM_Server.Step:= 23;
            END_IF

        23:
            SC_KOM_Server.StepName:= '23 - Priradenie QR kodu - odpoved servera';
            SC_KOM_Server.IdleTime.PT:= T#3s;
            SC_KOM_Server.AlarmTime.PT:= T#20s;
            SC_KOM_Server.AlarmTime.IN:= TRUE;

            IF SKTcpClientTrace_1.Status.staReceived AND
                (TRCB_P4_Vytah_ST10.OUTPUTS.TYP_Prikazu = TRCB_P4_Vytah_ST10.INPUTS.TYP_Prikazu) AND
                (TRCB_P4_Vytah_ST10.OUTPUTS.QRkodPowerCP = TRCB_P4_Vytah_ST10.INPUTS.QRkodPowerCP) THEN
                TRCB_P4_Vytah_ST10.STATUS.KomunikaciaUkoncena:= TRUE;
                SC_KOM_Server.ResetStep:= TRUE;
                SC_KOM_Server.Step:= 25;
            ELSIF SC_KOM_Server.AlarmTime.Q THEN
                TRCB_P4_Vytah_ST10.STATUS.KomunikaciaError:= TRUE;
                SC_KOM_Server.ResetStep:= TRUE;
                SC_KOM_Server.Step:= 25;
            END_IF

        25:
            SC_KOM_Server.StepName:= '25 - Vyziadanie stavu paletky - cakam na ukoncenie komunikacie';
            SC_KOM_Server.IdleTime.PT:= T#3s;
            SC_KOM_Server.AlarmTime.PT:= T#10s;

            IF NOT TRCB_P4_Vytah_ST10.CMD.PriradQRkodFiltra_TYP3 THEN
                SC_KOM_Server.ResetStep:= TRUE;
                SC_KOM_Server.Step:= 0;
            END_IF

        30:
            SC_KOM_Server.StepName:= '30 - Vyziadanie serioveho cisla - odoslanie dat na server';
            SC_KOM_Server.IdleTime.PT:= T#3s;
            SC_KOM_Server.AlarmTime.PT:= T#10s;

            TRCB_P4_Vytah_ST10.INPUTS.TYP_Prikazu:= '0';
            TRCB_P4_Vytah_ST10.INPUTS.CisloStanice:= 'ST10';
            TRCB_P4_Vytah_ST10.INPUTS.CisloPaletky;
            TRCB_P4_Vytah_ST10.INPUTS.QRkodPowerCP:= '';
            TRCB_P4_Vytah_ST10.INPUTS.QRkodFiltra:= '';
            TRCB_P4_Vytah_ST10.INPUTS.ID_Operatora:= 'E2';
            TRCB_P4_Vytah_ST10.INPUTS.Report:= '';
            TRCB_P4_Vytah_ST10.INPUTS.StavPaletky:= 'OK';
            SKTcpClientTrace_1.Cmd.Send:= TRUE;

            IF SKTcpClientTrace_1.Cmd.Send AND NOT SKTcpClientTrace_1.Status.staReceived AND NOT SKTcpClientTrace_1.Status.staError THEN
                SC_KOM_Server.ResetStep:= TRUE;
                SC_KOM_Server.Step:= 33;
            END_IF

        33:
            SC_KOM_Server.StepName:= '33 - Vyziadanie serioveho cisla - odpoved servera';
            SC_KOM_Server.IdleTime.PT:= T#3s;
            SC_KOM_Server.AlarmTime.PT:= T#20s;
            SC_KOM_Server.AlarmTime.IN:= TRUE;

            IF SKTcpClientTrace_1.Status.staReceived AND
                (TRCB_P4_Vytah_ST10.OUTPUTS.TYP_Prikazu = TRCB_P4_Vytah_ST10.INPUTS.TYP_Prikazu) THEN
                TRCB_P4_Vytah_ST10.STATUS.KomunikaciaUkoncena:= TRUE;
                SC_KOM_Server.ResetStep:= TRUE;
                SC_KOM_Server.Step:= 35;
            ELSIF SC_KOM_Server.AlarmTime.Q THEN
                TRCB_P4_Vytah_ST10.STATUS.KomunikaciaError:= TRUE;
                SC_KOM_Server.ResetStep:= TRUE;
                SC_KOM_Server.Step:= 35;
            END_IF

        35:
            SC_KOM_Server.StepName:= '35 - Vyziadanie serioveho cisla - cakam na ukoncenie komunikacie';
            SC_KOM_Server.IdleTime.PT:= T#3s;
            SC_KOM_Server.AlarmTime.PT:= T#10s;

            IF NOT TRCB_P4_Vytah_ST10.CMD.VyziadajCisloEtikety_TYP0 THEN
                SC_KOM_Server.ResetStep:= TRUE;
                SC_KOM_Server.Step:= 0;
            END_IF

        40:
            SC_KOM_Server.StepName:= '40 - Odoslanie stavu paletky - odoslanie dat na server';
            SC_KOM_Server.IdleTime.PT:= T#3s;
            SC_KOM_Server.AlarmTime.PT:= T#20s;
            SC_KOM_Server.AlarmTime.IN:= TRUE;

            IF NOT SC_KOM_Server.Switch1 THEN
                brsmemset(ADR(Report),0,SIZEOF(Report));
				brsmemset(ADR(TRCB_P4_Vytah_ST10.INPUTS.Report), 0, SIZEOF(TRCB_P4_Vytah_ST10.INPUTS.Report));

				//Kamera 16//
                Report[0].PoradoveCislo:= '1';
                Report[0].Popis:= 'KAM_16_KontrolaPaletky';
                Report[0].FormatHodnoty:= '2';
                Report[0].Tolerancia_MIN_Hodnota:= '';
                Report[0].Tolerancia_MAX_Hodnota:= '';
                Report[0].Nominal:= 'OK';
                Report[0].Tolerancia_MIN_Jednotky:= '';
                Report[0].Tolerancia_MAX_Jednotky:= '';
                IF Reports.Kamery.P4_CAM16_KontrolaPaletky = 'PASS' THEN
                    Report[0].NameranaHodnota:= 'OK';
                ELSE
                    Report[0].NameranaHodnota:= 'NG';
                END_IF
                Report[0].NameranaHodnota_Jednotky:= '';
                Report[0].VyslednyResult:= Reports.Kamery.P4_CAM16_KontrolaPaletky;
                SKTcpClientNewCsvEntry(Report[0].PoradoveCislo,Report[0].Popis,Report[0].FormatHodnoty,Report[0].Tolerancia_MIN_Hodnota,Report[0].Tolerancia_MAX_Hodnota,Report[0].Nominal,Report[0].Tolerancia_MIN_Jednotky,Report[0].Tolerancia_MAX_Jednotky,Report[0].NameranaHodnota,Report[0].NameranaHodnota_Jednotky,Report[0].VyslednyResult, ADR(TRCB_P4_Vytah_ST10.INPUTS.Report));
                SC_KOM_Server.Switch1:= TRUE;
            END_IF

            TRCB_P4_Vytah_ST10.INPUTS.TYP_Prikazu:= '2';
            TRCB_P4_Vytah_ST10.INPUTS.CisloStanice:= 'ST10';
            TRCB_P4_Vytah_ST10.INPUTS.CisloPaletky;
            TRCB_P4_Vytah_ST10.INPUTS.QRkodPowerCP:= Paletka[a].PAR.QRkodPowerCP;
            TRCB_P4_Vytah_ST10.INPUTS.QRkodFiltra:= '';
            TRCB_P4_Vytah_ST10.INPUTS.ID_Operatora:= Paletka[a].PAR.ID_Operatora;
            TRCB_P4_Vytah_ST10.INPUTS.Report:= '';
            TRCB_P4_Vytah_ST10.INPUTS.StavPaletky:= Paletka[a].PAR.StavPowerCP;
            SKTcpClientTrace_1.Cmd.Send:= TRUE;

            IF SKTcpClientTrace_1.Cmd.Send AND NOT SKTcpClientTrace_1.Status.staReceived AND NOT SKTcpClientTrace_1.Status.staError THEN
                SC_KOM_Server.ResetStep:= TRUE;
                SC_KOM_Server.Step:= 43;
            ELSIF SC_KOM_Server.AlarmTime.Q AND (SKTcpClientTrace_1.Status.staReceived OR SKTcpClientTrace_1.Status.staError) THEN
                PocetDopytovNaServer:= PocetDopytovNaServer + 1;
                SC_KOM_Server.ResetStep:= TRUE;
                SC_KOM_Server.Step:= 44;
            END_IF

        43:
            SC_KOM_Server.StepName:= '43 - Odoslanie stavu paletky - odpoved servera';
            SC_KOM_Server.IdleTime.PT:= T#3s;
            SC_KOM_Server.AlarmTime.PT:= T#20s;
            SC_KOM_Server.AlarmTime.IN:= TRUE;

            IF SKTcpClientTrace_1.Status.staReceived AND
                (TRCB_P4_Vytah_ST10.OUTPUTS.TYP_Prikazu = TRCB_P4_Vytah_ST10.INPUTS.TYP_Prikazu) AND
                (TRCB_P4_Vytah_ST10.OUTPUTS.QRkodPowerCP = TRCB_P4_Vytah_ST10.INPUTS.QRkodPowerCP) THEN
                TRCB_P4_Vytah_ST10.STATUS.KomunikaciaUkoncena:= TRUE;
                SC_KOM_Server.ResetStep:= TRUE;
                SC_KOM_Server.Step:= 45;
            ELSIF SC_KOM_Server.AlarmTime.Q THEN
                PocetDopytovNaServer:= PocetDopytovNaServer + 1;
                SC_KOM_Server.ResetStep:= TRUE;
                SC_KOM_Server.Step:= 44;
            END_IF

        44:
            SC_KOM_Server.StepName:= '44 - Odoslanie stavu paletky - cakam na opatovny dopyt na server';
            SC_KOM_Server.IdleTime.PT:= T#1s;
            SC_KOM_Server.AlarmTime.PT:= T#10s;
            SC_KOM_Server.IdleTime.IN:= TRUE;
            SKTcpClientTrace_1.Cmd.Send:= FALSE;

            IF PocetDopytovNaServer < 3 THEN
                IF SC_KOM_Server.IdleTime.Q THEN
                    SC_KOM_Server.ResetStep:= TRUE;
                    SC_KOM_Server.Step:= 40;
                END_IF
            ELSE
                TRCB_P4_Vytah_ST10.STATUS.KomunikaciaError:= TRUE;
                SC_KOM_Server.ResetStep:= TRUE;
                SC_KOM_Server.Step:= 45;
            END_IF

        45:
            SC_KOM_Server.StepName:= '45 - Vyziadanie serioveho cisla - cakam na ukoncenie komunikacie';
            SC_KOM_Server.IdleTime.PT:= T#3s;
            SC_KOM_Server.AlarmTime.PT:= T#10s;

            IF NOT TRCB_P4_Vytah_ST10.CMD.OdosliStavPaletky_TYP2 THEN
                SC_KOM_Server.ResetStep:= TRUE;
                SC_KOM_Server.Step:= 0;
            END_IF

    END_CASE

END_PROGRAM

PROGRAM _EXIT
	(* Insert code here *)

END_PROGRAM
```

#### Types.typ - Local data types
```iecst
TYPE
	Report_typ : 	STRUCT
		PoradoveCislo : STRING[2]; (*IDstep - Poradové čislo reportu*)
		Popis : STRING[100]; (*Description - Popis*)
		FormatHodnoty : STRING[2]; (*TypValue - Format zaslané hodnoty  1- Číslo, 2 - Znak*)
		Tolerancia_MIN_Hodnota : STRING[10]; (*MinTol - Minimálna tolerancia meranej veličiny*)
		Tolerancia_MAX_Hodnota : STRING[10]; (*MaxTol - Maximálna tolerancia meranej veličiny*)
		Nominal : STRING[10]; (*Nom - Ak jezvolený formát string tak tu zadáme OK inak je prazdna*)
		Tolerancia_MIN_Jednotky : STRING[10]; (*MinEle - Jednotky minimálnej tolerancie veličiny*)
		Tolerancia_MAX_Jednotky : STRING[10]; (*MaxEle - Jednotky maximálnej tolerancie veličiny*)
		NameranaHodnota : STRING[10]; (*Value - Namerana hodnota veličiny, ak su kamery tak bude hodnota OK alebo NG*)
		NameranaHodnota_Jednotky : STRING[10]; (*ValEle - Jednotky nameranej veličiny*)
		VyslednyResult : STRING[5]; (*Result - Výsledný result  PASS, FAIL, SKIP*)
	END_STRUCT;
END_TYPE
```

#### Variables.var - Local variables
```iecst
VAR
	SC_KOM_Server : SequenceControlTyp;
	SKTcpClientTrace_1 : SKTcpClientTrace;
	a : USINT;
	Report : ARRAY[0..50] OF Report_typ;
	PocetDopytovNaServer : USINT;
END_VAR
```

### Program Logical/RiadenieServ/RiadenieServ (IEC)

#### Main.st - Init, cyclic, exit code
```iecst
PROGRAM _INIT

	P1_Vytah.ServoZdvihuVytahu_M31.AxisName:= ADR(gAxis_6);
	P1_Srobovanie.ServoManipulOsX_M20.AxisName:= ADR(gAxis_7);
	P1_Srobovanie.ServoManipulOsY_M19.AxisName:= ADR(gAxis_8);
	P2_ZakladacTesnenia.ServoZdvihuZakladaca_M4.AxisName:= ADR(gAxis_1);
	P2_ZakladacTesnenia.ServoPojazduVozika_M5.AxisName:= ADR(gAxis_2);
	P2_Srobovanie.ServoManipulOsX_M10.AxisName:= ADR(gAxis_3);
	P2_Srobovanie.ServoManipulOsY_M9.AxisName:= ADR(gAxis_4);
	P2_Zvaranie.ServoZdvihuZvarania_M6.AxisName:= ADR(gAxis_5);
	P3_Srobovanie.ServoManipulOsY_M37.AxisName:= ADR(gAxis_9);
	P4_Vytah.ServoZdvihuVytahu_M26.AxisName:= ADR(gAxis_10);
	P4_Etiketovacka.ServoZdvihuEtiketovania_M28.AxisName:= ADR(gAxis_11);

END_PROGRAM

PROGRAM _CYCLIC

	//********************************************Pracovisko č.1*******************************************
	//Volanie funkcie//
	P1_Vytah.ServoZdvihuVytahu_M31();
	P1_Srobovanie.ServoManipulOsX_M20();
	P1_Srobovanie.ServoManipulOsY_M19();

	//P1 - vytah servo READY//
	IF (P1_Vytah.ServoZdvihuVytahu_M31.STATUS.Power_ON AND NOT P1_Vytah.ServoZdvihuVytahu_M31.STATUS.ERROR) THEN
		P1_Pracovisko.STAV.ServoVytahu_READY:= TRUE;
	ELSE
		P1_Pracovisko.STAV.ServoVytahu_READY:= FALSE;
	END_IF

	//P1 - status serva bunky READY//
	IF (P1_Vytah.ServoZdvihuVytahu_M31.STATUS.Power_ON AND NOT P1_Vytah.ServoZdvihuVytahu_M31.STATUS.ERROR) AND
		(P1_Srobovanie.ServoManipulOsX_M20.STATUS.Power_ON AND NOT P1_Srobovanie.ServoManipulOsX_M20.STATUS.ERROR) AND
		(P1_Srobovanie.ServoManipulOsY_M19.STATUS.Power_ON AND NOT P1_Srobovanie.ServoManipulOsY_M19.STATUS.ERROR) THEN
		P1_Pracovisko.STAV.ServaBunky_READY:= TRUE;
	ELSE
		P1_Pracovisko.STAV.ServaBunky_READY:= FALSE;
	END_IF

	//*********************************************Pracovisko č.2******************************************
	//Volanie funkcie//
	P2_ZakladacTesnenia.ServoZdvihuZakladaca_M4();
	P2_ZakladacTesnenia.ServoPojazduVozika_M5();
	P2_Srobovanie.ServoManipulOsX_M10();
	P2_Srobovanie.ServoManipulOsY_M9();
	P2_Zvaranie.ServoZdvihuZvarania_M6();

	//P2 - status serva zakladača READY//
	IF (P2_ZakladacTesnenia.ServoZdvihuZakladaca_M4.STATUS.Power_ON AND NOT P2_ZakladacTesnenia.ServoZdvihuZakladaca_M4.STATUS.ERROR) AND
		(P2_ZakladacTesnenia.ServoPojazduVozika_M5.STATUS.Power_ON AND NOT P2_ZakladacTesnenia.ServoPojazduVozika_M5.STATUS.ERROR) THEN
		P2_Pracovisko.STAV.ServaZakladaca_READY:= TRUE;
	ELSE
		P2_Pracovisko.STAV.ServaZakladaca_READY:= FALSE;
	END_IF

	//P2 - status serva bunky READY//
	IF (P2_Srobovanie.ServoManipulOsX_M10.STATUS.Power_ON AND NOT P2_Srobovanie.ServoManipulOsX_M10.STATUS.ERROR) AND
		(P2_Srobovanie.ServoManipulOsY_M9.STATUS.Power_ON AND NOT P2_Srobovanie.ServoManipulOsY_M9.STATUS.ERROR) AND
		(P2_Zvaranie.ServoZdvihuZvarania_M6.STATUS.Power_ON AND NOT P2_Zvaranie.ServoZdvihuZvarania_M6.STATUS.ERROR) THEN
		P2_Pracovisko.STAV.ServaBunky_READY:= TRUE;
	ELSE
		P2_Pracovisko.STAV.ServaBunky_READY:= FALSE;
	END_IF

	//********************************************Pracovisko č.3*******************************************
	//Volanie funkcie//
	P3_Srobovanie.ServoManipulOsY_M37();

	//P3 - status serva bunky READY//
	IF (P3_Srobovanie.ServoManipulOsY_M37.STATUS.Power_ON AND NOT P3_Srobovanie.ServoManipulOsY_M37.STATUS.ERROR) THEN
		P3_Pracovisko.STAV.ServaBunky_READY:= TRUE;
	ELSE
		P3_Pracovisko.STAV.ServaBunky_READY:= FALSE;
	END_IF

	//********************************************Pracovisko č.4*******************************************
	//Volanie funkcie//
	P4_Vytah.ServoZdvihuVytahu_M26();
	P4_Etiketovacka.ServoZdvihuEtiketovania_M28();

	//P4 - vytah servo READY//
	IF (P4_Vytah.ServoZdvihuVytahu_M26.STATUS.Power_ON AND NOT P4_Vytah.ServoZdvihuVytahu_M26.STATUS.ERROR) THEN
		P4_Pracovisko.STAV.ServoVytahu_READY:= TRUE;
	ELSE
		P4_Pracovisko.STAV.ServoVytahu_READY:= FALSE;
	END_IF

	//P4 - status serva bunky READY//
	IF (P4_Etiketovacka.ServoZdvihuEtiketovania_M28.STATUS.Power_ON AND NOT P4_Etiketovacka.ServoZdvihuEtiketovania_M28.STATUS.ERROR) THEN
		P4_Pracovisko.STAV.ServaBunky_READY:= TRUE;
	ELSE
		P4_Pracovisko.STAV.ServaBunky_READY:= FALSE;
	END_IF

END_PROGRAM

PROGRAM _EXIT
	(* Insert code here *)

END_PROGRAM
```

### Program Logical/RiadenieServ/LimitneSnimace (IEC)

#### Main.st - Init, cyclic, exit code
```iecst
PROGRAM _INIT
	(* Insert code here *)

END_PROGRAM

PROGRAM _CYCLIC
	//ENABLE pre limitné snímače sa musí spustiť pred Power serva//

	//************************P1 - Výtah********************************//
	//Servo zdvihu výťahu//
	IF P1_Vytah.ServoZdvihuVytahu_M31.STATUS.Communication_READY THEN
		ServoLimSnimace_5.ENABLE:= TRUE;
	ELSE
		ServoLimSnimace_5.ENABLE:= FALSE;
	END_IF
	ServoLimSnimace_5.AxisName:= ADR(gAxis_6);
	P1_Vytah.STAV.ServoZvihu_LimitSnimace_BUSY:= ServoLimSnimace_5.BUSY;
	ServoLimSnimace_5.HomingSwitch;
	ServoLimSnimace_5.NegativeLimitSwitch:= P1_Vytah.IN.ZdvihVytahu_LimSnimacNEG_IS60;
	ServoLimSnimace_5.PositiveLimitSwitch:= P1_Vytah.IN.ZdvihVytahu_LimSnimacPOS_IS61;
	ServoLimSnimace_5();

	//***************************P1 - Srobovanie********************************//
	//Servo - pojazd manipulátora Os X//
	IF P1_Srobovanie.ServoManipulOsX_M20.STATUS.Communication_READY THEN
		ServoLimSnimace_6.ENABLE:= TRUE;
	ELSE
		ServoLimSnimace_6.ENABLE:= FALSE;
	END_IF
	ServoLimSnimace_6.AxisName:= ADR(gAxis_7);
	P1_Srobovanie.STAV.OsX_LimitSnimace_BUSY:= ServoLimSnimace_6.BUSY;
	ServoLimSnimace_6.HomingSwitch;
	ServoLimSnimace_6.NegativeLimitSwitch:= P1_Srobovanie.IN.ManipulOsX_LimSnimacPOS_IS43;
	ServoLimSnimace_6.PositiveLimitSwitch:= P1_Srobovanie.IN.ManipulOsX_LimSnimacNEG_IS42;
	ServoLimSnimace_6();

	//Servo - pojazd manipulatora Os Y//
	IF P1_Srobovanie.ServoManipulOsY_M19.STATUS.Communication_READY THEN
		ServoLimSnimace_7.ENABLE:= TRUE;
	ELSE
		ServoLimSnimace_7.ENABLE:= FALSE;
	END_IF
	ServoLimSnimace_7.AxisName:= ADR(gAxis_8);
	P1_Srobovanie.STAV.OsY_LimitSnimace_BUSY:= ServoLimSnimace_7.BUSY;
	ServoLimSnimace_7.HomingSwitch;
	ServoLimSnimace_7.NegativeLimitSwitch:= P1_Srobovanie.IN.ManipulOsY_LimSnimacPOS_IS41;
	ServoLimSnimace_7.PositiveLimitSwitch:= P1_Srobovanie.IN.ManipulOsY_LimSnimacNEG_IS40;
	ServoLimSnimace_7();

	//***************************P2 - Zakladač tesnenia ******************//
	//Servo - zdvihu//
	IF P2_ZakladacTesnenia.ServoZdvihuZakladaca_M4.STATUS.Communication_READY THEN
		ServoLimSnimace_0.ENABLE:= TRUE;
	ELSE
		ServoLimSnimace_0.ENABLE:= FALSE;
	END_IF
	ServoLimSnimace_0.AxisName:= ADR(gAxis_1);
	P2_ZakladacTesnenia.STAV.ServoZvihu_LimitSnimace_BUSY:= ServoLimSnimace_0.BUSY;
	ServoLimSnimace_0.HomingSwitch:= P2_ZakladacTesnenia.IN.ZdvihZaklad_RefSnimac_IS8;
	ServoLimSnimace_0.NegativeLimitSwitch;
	ServoLimSnimace_0.PositiveLimitSwitch;
	ServoLimSnimace_0();

	//Servo - pojazdu//
	IF P2_ZakladacTesnenia.ServoPojazduVozika_M5.STATUS.Communication_READY THEN
		ServoLimSnimace_1.ENABLE:= TRUE;
	ELSE
		ServoLimSnimace_1.ENABLE:= FALSE;
	END_IF
	ServoLimSnimace_1.AxisName:= ADR(gAxis_2);
	P2_ZakladacTesnenia.STAV.ServoPojazdu_LimitSnimace_BUSY:= ServoLimSnimace_1.BUSY;
	ServoLimSnimace_1.HomingSwitch;
	ServoLimSnimace_1.NegativeLimitSwitch;
	ServoLimSnimace_1.PositiveLimitSwitch;
	ServoLimSnimace_1();

	//***************************P2 - Srobovanie********************************//
	//Servo - pojazd manipulátora Os X//
	IF P2_Srobovanie.ServoManipulOsX_M10.STATUS.Communication_READY THEN
		ServoLimSnimace_2.ENABLE:= TRUE;
	ELSE
		ServoLimSnimace_2.ENABLE:= FALSE;
	END_IF
	ServoLimSnimace_2.AxisName:= ADR(gAxis_3);
	P2_Srobovanie.STAV.OsX_LimitSnimace_BUSY:= ServoLimSnimace_2.BUSY;
	ServoLimSnimace_2.HomingSwitch;
	ServoLimSnimace_2.NegativeLimitSwitch:= P2_Srobovanie.IN.ManipulOsX_LimSnimacNEG_IS22;
	ServoLimSnimace_2.PositiveLimitSwitch:= P2_Srobovanie.IN.ManipulOsX_LimSnimacPOS_IS21;
	ServoLimSnimace_2();

	//Servo - pojazd manipulatora Os Y//
	IF P2_Srobovanie.ServoManipulOsY_M9.STATUS.Communication_READY THEN
		ServoLimSnimace_3.ENABLE:= TRUE;
	ELSE
		ServoLimSnimace_3.ENABLE:= FALSE;
	END_IF
	ServoLimSnimace_3.AxisName:= ADR(gAxis_4);
	P2_Srobovanie.STAV.OsY_LimitSnimace_BUSY:= ServoLimSnimace_3.BUSY;
	ServoLimSnimace_3.HomingSwitch;
	ServoLimSnimace_3.NegativeLimitSwitch:= P2_Srobovanie.IN.ManipulOsY_LimSnimacNEG_IS20;
	ServoLimSnimace_3.PositiveLimitSwitch:= P2_Srobovanie.IN.ManipulOsY_LimSnimacPOS_IS19;
	ServoLimSnimace_3();

	//*****************************P2 Zváranie************************************//
	//Servo zdvihu zvárania//
	IF P2_Zvaranie.ServoZdvihuZvarania_M6.STATUS.Communication_READY THEN
		ServoLimSnimace_4.ENABLE:= TRUE;
	ELSE
		ServoLimSnimace_4.ENABLE:= FALSE;
	END_IF
	ServoLimSnimace_4.AxisName:= ADR(gAxis_5);
	P2_Zvaranie.STAV.ServoZvihu_LimitSnimace_BUSY:= ServoLimSnimace_4.BUSY;
	ServoLimSnimace_4.HomingSwitch:= P2_Zvaranie.IN.ZdvihZvarania_RefSnimac_IS9;
	ServoLimSnimace_4.NegativeLimitSwitch;
	ServoLimSnimace_4.PositiveLimitSwitch;
	ServoLimSnimace_4();

	//***************************P3 - Srobovanie********************************//
	//Servo - pojazd manipulatora Os Y//
	IF P3_Srobovanie.ServoManipulOsY_M37.STATUS.Communication_READY THEN
		ServoLimSnimace_8.ENABLE:= TRUE;
	ELSE
		ServoLimSnimace_8.ENABLE:= FALSE;
	END_IF
	ServoLimSnimace_8.AxisName:= ADR(gAxis_9);
	P3_Srobovanie.STAV.OsY_LimitSnimace_BUSY:= ServoLimSnimace_8.BUSY;
	ServoLimSnimace_8.HomingSwitch;
	ServoLimSnimace_8.NegativeLimitSwitch:= P3_Srobovanie.IN.ManipulOsY_LimSnimacNEG_IS76;
	ServoLimSnimace_8.PositiveLimitSwitch:= P3_Srobovanie.IN.ManipulOsY_LimSnimacPOS_IS75;
	ServoLimSnimace_8();

	//***************************P4 - Vytah***************************************//
	//Servo zdvihu výťahu//
	IF P4_Vytah.ServoZdvihuVytahu_M26.STATUS.Communication_READY THEN
		ServoLimSnimace_9.ENABLE:= TRUE;
	ELSE
		ServoLimSnimace_9.ENABLE:= FALSE;
	END_IF
	ServoLimSnimace_9.AxisName:= ADR(gAxis_10);
	P4_Vytah.STAV.ServoZvihu_LimitSnimace_BUSY:= ServoLimSnimace_9.BUSY;
	ServoLimSnimace_9.HomingSwitch;
	ServoLimSnimace_9.NegativeLimitSwitch:= P4_Vytah.IN.ZdvihVytahu_LimSnimacNEG_IS56;
	ServoLimSnimace_9.PositiveLimitSwitch:= P4_Vytah.IN.ZdvihVytahu_LimSnimacPOS_IS57;
	ServoLimSnimace_9();

	//****************************P4 - Etiketovanie*****************************//
	//Servo zdvihu etiketovania//
	IF P4_Etiketovacka.ServoZdvihuEtiketovania_M28.STATUS.Communication_READY THEN
		ServoLimSnimace_10.ENABLE:= TRUE;
	ELSE
		ServoLimSnimace_10.ENABLE:= FALSE;
	END_IF
	ServoLimSnimace_10.AxisName:= ADR(gAxis_11);
	P4_Etiketovacka.STAV.ServoZvihu_LimitSnimace_BUSY:= ServoLimSnimace_10.BUSY;
	ServoLimSnimace_10.HomingSwitch:= P4_Etiketovacka.IN.ZdvihEtiketovania_RefSnimac_IS59;
	ServoLimSnimace_10.NegativeLimitSwitch;
	ServoLimSnimace_10.PositiveLimitSwitch;
	ServoLimSnimace_10();

END_PROGRAM

PROGRAM _EXIT
	(* Insert code here *)

END_PROGRAM
```

#### Variables.var - Local variables
```iecst
VAR
	ServoLimSnimace_0 : ServoLim;
	ServoLimSnimace_1 : ServoLim;
	ServoLimSnimace_2 : ServoLim;
	ServoLimSnimace_3 : ServoLim;
	ServoLimSnimace_4 : ServoLim;
	ServoLimSnimace_5 : ServoLim;
	ServoLimSnimace_6 : ServoLim;
	ServoLimSnimace_7 : ServoLim;
	ServoLimSnimace_8 : ServoLim;
	ServoLimSnimace_9 : ServoLim;
	ServoLimSnimace_10 : ServoLim;
END_VAR
```

### Program Logical/RemanentnePremenne/P1_RemanentnePremenne (IEC)

#### Main.st - Init, cyclic, exit code
```iecst
PROGRAM _INIT
	(* Insert code here *)

END_PROGRAM

PROGRAM _CYCLIC

	P1_RemPremenne;

	//Načítanie premenných pri prvom spustení//
	IF EDGEPOS(Safety.STAV.SafetyPLC_Nabehlo) THEN
		P1_NacitajPremenne:= TRUE;
	END_IF

	//Načítanie premenných z pamäte//
	IF P1_NacitajPremenne THEN
		MpRecipeXml_P1.Load:= TRUE;
		P1_NacitajPremenne:= FALSE;
	END_IF

	IF MpRecipeXml_P1.Load AND (MpRecipeXml_P1.CommandDone OR MpRecipeXml_P1.Error) THEN
		MpRecipeXml_P1.Load:= FALSE;
	END_IF

	//Konfigurácia premenných//
	MpRecipeXml_P1.MpLink:= ADR(gRemPremenneP1);  //takto sa menuje mapp komponenta v configurating view//
	MpRecipeXml_P1.Enable:= TRUE;
	MpRecipeXml_P1.Category:= ADR('PREMENNE_P1');
	MpRecipeXml_P1.DeviceName:= ADR('HDD_RemPremenneP1');  //Názov media, kde sa budú receptury ukladat//
	MpRecipeXml_P1.FileName:= ADR('RemPremenneP1'); //Názov súboru do ktorého sa receptúry uložia//
	MpRecipeXml_P1();

	MpRecipeRegPar_P1.MpLink:= ADR(gRemPremenneP1);
	MpRecipeRegPar_P1.Enable:= TRUE;
	MpRecipeRegPar_P1.Category:= ADR('PREMENNE_P1');
	MpRecipeRegPar_P1.PVName:= ADR('P1_RemPremenne'); //Názov premenné, kde je vytvorená štruktura dat premennych//
	MpRecipeRegPar_P1();

	//Uloženie premenných//
	IF P1_UlozPremenne THEN
		MpRecipeXml_P1.Save:= TRUE;
		P1_UlozPremenne:= FALSE;
	END_IF

	IF MpRecipeXml_P1.Save AND (MpRecipeXml_P1.CommandDone OR MpRecipeXml_P1.Error) THEN
		MpRecipeXml_P1.Save:= FALSE;
	END_IF

END_PROGRAM

PROGRAM _EXIT
	(* Insert code here *)

END_PROGRAM
```

#### Variables.var - Local variables
```iecst
VAR
	UISetup : MpRecipeUISetupType;
	UIConnect : MpRecipeUIConnectType := (0);
END_VAR
```

### Program Logical/RemanentnePremenne/P2_RemanentnePremenne (IEC)

#### Main.st - Init, cyclic, exit code
```iecst
PROGRAM _INIT

END_PROGRAM

PROGRAM _CYCLIC

	P2_RemPremenne;

	//Načítanie premenných pri prvom spustení//
	IF EDGEPOS(Safety.STAV.SafetyPLC_Nabehlo) THEN
		P2_NacitajPremenne:= TRUE;
	END_IF

	//Načítanie premenných z pamäte//
	IF P2_NacitajPremenne THEN
		MpRecipeXml_P2.Load:= TRUE;
		P2_NacitajPremenne:= FALSE;
	END_IF

	IF MpRecipeXml_P2.Load AND (MpRecipeXml_P2.CommandDone OR MpRecipeXml_P2.Error) THEN
		MpRecipeXml_P2.Load:= FALSE;
	END_IF

	//Konfigurácia premenných//
	MpRecipeXml_P2.MpLink:= ADR(gRemPremenneP2);  //takto sa menuje mapp komponenta v configurating view//
	MpRecipeXml_P2.Enable:= TRUE;
	MpRecipeXml_P2.Category:= ADR('PREMENNE_P2');
	MpRecipeXml_P2.DeviceName:= ADR('HDD_RemPremenneP2');  //Názov media, kde sa budú receptury ukladat//
	MpRecipeXml_P2.FileName:= ADR('RemPremenneP2'); //Názov súboru do ktorého sa receptúry uložia//
	MpRecipeXml_P2();

	MpRecipeRegPar_P2.MpLink:= ADR(gRemPremenneP2);
	MpRecipeRegPar_P2.Enable:= TRUE;
	MpRecipeRegPar_P2.Category:= ADR('PREMENNE_P2');
	MpRecipeRegPar_P2.PVName:= ADR('P2_RemPremenne'); //Názov premenné, kde je vytvorená štruktura dat premenných//
	MpRecipeRegPar_P2();

	//Uloženie premenných//
	IF P2_UlozPremenne THEN
		MpRecipeXml_P2.Save:= TRUE;
		P2_UlozPremenne:= FALSE;
	END_IF

	IF MpRecipeXml_P2.Save AND (MpRecipeXml_P2.CommandDone OR MpRecipeXml_P2.Error) THEN
		MpRecipeXml_P2.Save:= FALSE;
	END_IF

END_PROGRAM

PROGRAM _EXIT
	(* Insert code here *)

END_PROGRAM
```

#### Variables.var - Local variables
```iecst
VAR
	UISetup : MpRecipeUISetupType;
	UIConnect : MpRecipeUIConnectType := (0);
END_VAR
```

### Program Logical/RemanentnePremenne/P34_RemanentnePremenne (IEC)

#### Main.st - Init, cyclic, exit code
```iecst
PROGRAM _INIT
	(* Insert code here *)

END_PROGRAM

PROGRAM _CYCLIC

	P34_RemPremenne;
	//Načítanie premenných pri prvom spustení//
	IF EDGEPOS(Safety.STAV.SafetyPLC_Nabehlo) THEN
		P34_NacitajPremenne:= TRUE;
	END_IF

	//Načítanie premenných z pamäte//
	IF P34_NacitajPremenne THEN
		MpRecipeXml_P34.Load:= TRUE;
		P34_NacitajPremenne:= FALSE;
	END_IF

	IF MpRecipeXml_P34.Load AND (MpRecipeXml_P34.CommandDone OR MpRecipeXml_P34.Error) THEN
		MpRecipeXml_P34.Load:= FALSE;
	END_IF

	//Konfigurácia premenných//
	MpRecipeXml_P34.MpLink:= ADR(gRemPremenneP34);  //takto sa menuje mapp komponenta v configurating view//
	MpRecipeXml_P34.Enable:= TRUE;
	MpRecipeXml_P34.Category:= ADR('PREMENNE_P34');
	MpRecipeXml_P34.DeviceName:= ADR('HDD_RemPremenneP34');  //Názov media, kde sa budú receptury ukladat//
	MpRecipeXml_P34.FileName:= ADR('RemPremenneP34'); //Názov súboru do ktorého sa receptúry uložia//
	MpRecipeXml_P34();

	MpRecipeRegPar_P34.MpLink:= ADR(gRemPremenneP34);
	MpRecipeRegPar_P34.Enable:= TRUE;
	MpRecipeRegPar_P34.Category:= ADR('PREMENNE_P34');
	MpRecipeRegPar_P34.PVName:= ADR('P34_RemPremenne'); //Názov premenné, kde je vytvorená štruktura dat premennych//
	MpRecipeRegPar_P34();

	//Uloženie premenných//
	IF P34_UlozPremenne THEN
		MpRecipeXml_P34.Save:= TRUE;
		P34_UlozPremenne:= FALSE;
	END_IF

	IF MpRecipeXml_P34.Save AND (MpRecipeXml_P34.CommandDone OR MpRecipeXml_P34.Error) THEN
		MpRecipeXml_P34.Save:= FALSE;
	END_IF

END_PROGRAM

PROGRAM _EXIT
	(* Insert code here *)

END_PROGRAM
```

#### Variables.var - Local variables
```iecst
VAR
	UISetup : MpRecipeUISetupType;
	UIConnect : MpRecipeUIConnectType := (0);
END_VAR
```

### Program Logical/OdosielanieFotiek/FTP_CAM1 (IEC)
